Yaskawa INFORM job: A_ROOF_SIDE_0617_2_PAINT_2.JBI

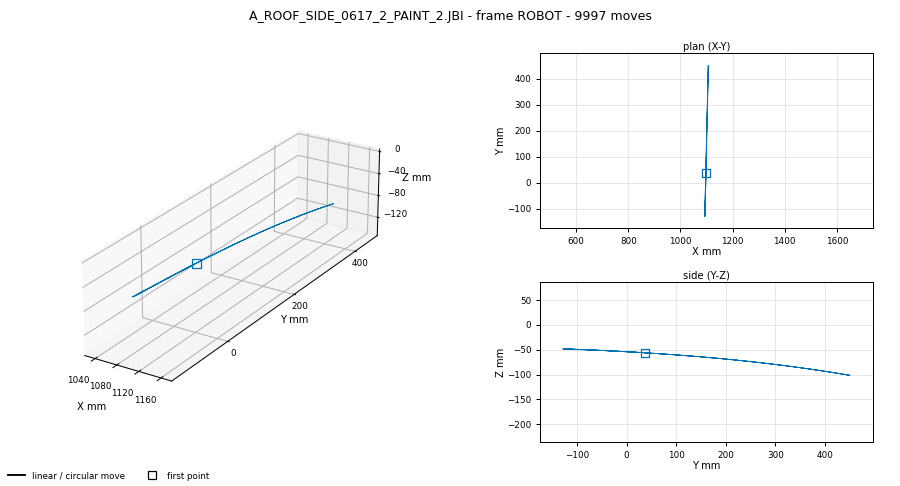
[picture p0: tool path of A_ROOF_SIDE_0617_2_PAINT_2.JBI in frame ROBOT, 9997 of 9997 moves have a stored position in this frame; points joined in program order, loops and branches not executed]
/JOB
//NAME A_ROOF_SIDE_0617_2_PAINT2
//POS
///NPOS 9997,0,0,0,0,0
///TOOL 1
///USER 0
///POSTYPE ROBOT
///RECTAN
///RCONF 1,0,0,0,0,0,0,0,0,0,0,0,0,0,0,0,0,0,0,0,0,0,0,0
C00000=1098.376,37.248,-55.821,176.207,15.311,152.033
C00001=1098.370,36.999,-55.805,176.206,15.311,152.033
C00002=1098.365,36.749,-55.790,176.204,15.310,152.034
C00003=1098.358,36.500,-55.775,176.201,15.310,152.034
C00004=1098.353,36.250,-55.760,176.199,15.308,152.034
C00005=1098.347,36.001,-55.745,176.197,15.308,152.035
C00006=1098.341,35.751,-55.729,176.195,15.307,152.035
C00007=1098.336,35.502,-55.713,176.192,15.306,152.035
C00008=1098.329,35.252,-55.698,176.190,15.306,152.036
C00009=1098.324,35.003,-55.683,176.188,15.305,152.036
C00010=1098.318,34.753,-55.668,176.185,15.304,152.036
C00011=1098.312,34.503,-55.653,176.183,15.303,152.037
C00012=1098.307,34.255,-55.638,176.181,15.303,152.037
C00013=1098.301,34.005,-55.623,176.178,15.302,152.037
C00014=1098.296,33.755,-55.607,176.176,15.301,152.038
C00015=1098.289,33.506,-55.593,176.174,15.301,152.038
C00016=1098.284,33.256,-55.577,176.172,15.300,152.038
C00017=1098.278,33.007,-55.562,176.170,15.299,152.038
C00018=1098.273,32.758,-55.547,176.167,15.298,152.039
C00019=1098.266,32.508,-55.532,176.166,15.298,152.039
C00020=1098.261,32.258,-55.516,176.163,15.296,152.039
C00021=1098.254,31.985,-55.500,176.161,15.296,152.040
C00022=1098.248,31.711,-55.483,176.158,15.295,152.040
C00023=1098.242,31.437,-55.466,176.156,15.294,152.041
C00024=1098.236,31.164,-55.450,176.153,15.293,152.041
C00025=1098.230,30.914,-55.435,176.151,15.292,152.041
C00026=1098.224,30.665,-55.420,176.149,15.292,152.041
C00027=1098.218,30.415,-55.405,176.147,15.291,152.042
C00028=1098.213,30.166,-55.390,176.145,15.290,152.042
C00029=1098.207,29.916,-55.375,176.142,15.290,152.042
C00030=1098.202,29.667,-55.361,176.140,15.288,152.043
C00031=1098.196,29.417,-55.345,176.138,15.288,152.043
C00032=1098.190,29.168,-55.331,176.136,15.287,152.043
C00033=1098.185,28.918,-55.315,176.134,15.287,152.044
C00034=1098.179,28.669,-55.301,176.131,15.285,152.044
C00035=1098.172,28.419,-55.286,176.129,15.285,152.044
C00036=1098.167,28.170,-55.270,176.127,15.284,152.045
C00037=1098.161,27.920,-55.255,176.124,15.283,152.045
C00038=1098.156,27.671,-55.240,176.123,15.282,152.045
C00039=1098.149,27.421,-55.225,176.121,15.281,152.045
C00040=1098.144,27.172,-55.211,176.118,15.281,152.046
C00041=1098.138,26.922,-55.196,176.116,15.280,152.046
C00042=1098.133,26.673,-55.181,176.114,15.279,152.046
C00043=1098.126,26.423,-55.166,176.112,15.278,152.047
C00044=1098.121,26.174,-55.151,176.110,15.278,152.047
C00045=1098.115,25.925,-55.137,176.107,15.277,152.047
C00046=1098.109,25.675,-55.122,176.105,15.276,152.048
C00047=1098.104,25.425,-55.107,176.103,15.275,152.048
C00048=1098.098,25.176,-55.092,176.100,15.274,152.048
C00049=1098.092,24.927,-55.078,176.099,15.274,152.049
C00050=1098.086,24.677,-55.062,176.097,15.273,152.049
C00051=1098.081,24.427,-55.048,176.095,15.272,152.049
C00052=1098.075,24.178,-55.033,176.092,15.271,152.049
C00053=1098.069,23.929,-55.019,176.090,15.271,152.050
C00054=1098.063,23.679,-55.003,176.088,15.270,152.050
C00055=1098.058,23.429,-54.989,176.086,15.269,152.050
C00056=1098.052,23.180,-54.975,176.084,15.268,152.051
C00057=1098.046,22.930,-54.959,176.081,15.268,152.051
C00058=1098.040,22.681,-54.945,176.080,15.267,152.051
C00059=1098.034,22.431,-54.930,176.077,15.265,152.051
C00060=1098.029,22.182,-54.916,176.075,15.265,152.052
C00061=1098.024,21.933,-54.901,176.073,15.264,152.052
C00062=1098.017,21.682,-54.886,176.071,15.264,152.052
C00063=1098.012,21.434,-54.872,176.068,15.262,152.053
C00064=1098.005,21.184,-54.857,176.066,15.262,152.053
C00065=1098.001,20.934,-54.842,176.064,15.261,152.053
C00066=1097.995,20.685,-54.828,176.063,15.260,152.053
C00067=1097.988,20.435,-54.813,176.060,15.259,152.054
C00068=1097.983,20.186,-54.799,176.058,15.258,152.054
C00069=1097.978,19.937,-54.784,176.056,15.258,152.054
C00070=1097.972,19.687,-54.769,176.054,15.257,152.055
C00071=1097.966,19.437,-54.755,176.051,15.256,152.055
C00072=1097.960,19.188,-54.740,176.049,15.255,152.055
C00073=1097.954,18.938,-54.726,176.048,15.254,152.055
C00074=1097.948,18.689,-54.712,176.046,15.254,152.056
C00075=1097.942,18.439,-54.697,176.043,15.253,152.056
C00076=1097.937,18.190,-54.682,176.041,15.252,152.056
C00077=1097.932,17.941,-54.668,176.039,15.251,152.057
C00078=1097.925,17.690,-54.653,176.037,15.251,152.057
C00079=1097.920,17.441,-54.639,176.034,15.249,152.057
C00080=1097.914,17.192,-54.625,176.033,15.248,152.057
C00081=1097.908,16.942,-54.610,176.031,15.248,152.058
C00082=1097.902,16.693,-54.596,176.028,15.247,152.058
C00083=1097.897,16.444,-54.582,176.026,15.246,152.058
C00084=1097.891,16.193,-54.567,176.024,15.245,152.059
C00085=1097.884,15.922,-54.551,176.022,15.245,152.059
C00086=1097.878,15.649,-54.535,176.019,15.243,152.059
C00087=1097.872,15.376,-54.520,176.017,15.243,152.059
C00088=1097.866,15.104,-54.505,176.015,15.241,152.060
C00089=1097.859,14.854,-54.490,176.013,15.241,152.060
C00090=1097.855,14.605,-54.475,176.011,15.240,152.060
C00091=1097.849,14.356,-54.461,176.009,15.240,152.061
C00092=1097.843,14.106,-54.447,176.006,15.238,152.061
C00093=1097.837,13.856,-54.432,176.004,15.237,152.061
C00094=1097.831,13.607,-54.419,176.002,15.237,152.061
C00095=1097.825,13.358,-54.404,176.001,15.236,152.062
C00096=1097.819,13.108,-54.390,175.999,15.235,152.062
C00097=1097.814,12.858,-54.376,175.996,15.234,152.062
C00098=1097.808,12.609,-54.361,175.994,15.234,152.063
C00099=1097.802,12.359,-54.347,175.992,15.233,152.063
C00100=1097.796,12.110,-54.333,175.990,15.232,152.063
C00101=1097.790,11.861,-54.319,175.987,15.231,152.064
C00102=1097.784,11.610,-54.304,175.986,15.230,152.064
C00103=1097.779,11.361,-54.290,175.984,15.229,152.064
C00104=1097.773,11.112,-54.276,175.982,15.229,152.064
C00105=1097.767,10.862,-54.261,175.980,15.228,152.065
C00106=1097.761,10.613,-54.247,175.977,15.227,152.065
C00107=1097.755,10.363,-54.234,175.975,15.226,152.065
C00108=1097.749,10.114,-54.219,175.973,15.225,152.065
C00109=1097.743,9.864,-54.205,175.971,15.225,152.066
C00110=1097.738,9.614,-54.191,175.969,15.224,152.066
C00111=1097.732,9.365,-54.177,175.967,15.223,152.066
C00112=1097.726,9.115,-54.162,175.965,15.222,152.067
C00113=1097.720,8.866,-54.149,175.963,15.221,152.067
C00114=1097.715,8.616,-54.135,175.961,15.221,152.067
C00115=1097.708,8.367,-54.121,175.958,15.219,152.067
C00116=1097.702,8.117,-54.107,175.957,15.219,152.068
C00117=1097.697,7.868,-54.093,175.955,15.218,152.068
C00118=1097.691,7.618,-54.079,175.953,15.217,152.068
C00119=1097.685,7.369,-54.064,175.951,15.216,152.068
C00120=1097.679,7.119,-54.050,175.948,15.215,152.069
C00121=1097.674,6.869,-54.036,175.946,15.214,152.069
C00122=1097.668,6.620,-54.023,175.944,15.214,152.069
C00123=1097.662,6.370,-54.009,175.943,15.213,152.069
C00124=1097.656,6.121,-53.994,175.941,15.212,152.070
C00125=1097.650,5.871,-53.980,175.938,15.211,152.070
C00126=1097.645,5.622,-53.966,175.936,15.210,152.070
C00127=1097.639,5.372,-53.952,175.934,15.209,152.070
C00128=1097.633,5.123,-53.939,175.932,15.209,152.071
C00129=1097.627,4.874,-53.925,175.931,15.208,152.071
C00130=1097.621,4.623,-53.910,175.928,15.207,152.071
C00131=1097.616,4.374,-53.896,175.926,15.206,152.072
C00132=1097.610,4.124,-53.883,175.924,15.205,152.072
C00133=1097.604,3.875,-53.869,175.922,15.204,152.072
C00134=1097.599,3.625,-53.855,175.920,15.204,152.072
C00135=1097.593,3.376,-53.842,175.918,15.202,152.073
C00136=1097.588,3.126,-53.828,175.916,15.202,152.073
C00137=1097.581,2.877,-53.813,175.914,15.201,152.073
C00138=1097.575,2.627,-53.800,175.912,15.200,152.073
C00139=1097.570,2.378,-53.786,175.910,15.199,152.073
C00140=1097.564,2.128,-53.772,175.908,15.198,152.074
C00141=1097.559,1.879,-53.758,175.906,15.197,152.074
C00142=1097.553,1.629,-53.745,175.904,15.196,152.074
C00143=1097.547,1.380,-53.731,175.902,15.195,152.075
C00144=1097.541,1.130,-53.717,175.900,15.195,152.075
C00145=1097.536,0.880,-53.703,175.898,15.194,152.075
C00146=1097.529,0.631,-53.689,175.896,15.193,152.075
C00147=1097.524,0.381,-53.676,175.894,15.192,152.076
C00148=1097.518,0.132,-53.662,175.892,15.191,152.076
C00149=1097.512,-0.139,-53.646,175.890,15.190,152.076
C00150=1097.506,-0.409,-53.632,175.887,15.189,152.076
C00151=1097.500,-0.679,-53.617,175.886,15.188,152.077
C00152=1097.493,-0.949,-53.602,175.884,15.188,152.077
C00153=1097.488,-1.199,-53.589,175.881,15.186,152.077
C00154=1097.482,-1.448,-53.575,175.879,15.185,152.077
C00155=1097.476,-1.699,-53.560,175.878,15.184,152.078
C00156=1097.470,-1.948,-53.547,175.876,15.184,152.078
C00157=1097.465,-2.198,-53.534,175.874,15.183,152.078
C00158=1097.459,-2.448,-53.520,175.871,15.182,152.078
C00159=1097.454,-2.697,-53.506,175.869,15.181,152.079
C00160=1097.448,-2.946,-53.493,175.867,15.180,152.079
C00161=1097.442,-3.196,-53.479,175.866,15.179,152.079
C00162=1097.437,-3.446,-53.465,175.864,15.178,152.079
C00163=1097.431,-3.695,-53.452,175.862,15.177,152.079
C00164=1097.425,-3.944,-53.438,175.859,15.176,152.080
C00165=1097.419,-4.194,-53.425,175.858,15.175,152.080
C00166=1097.413,-4.443,-53.411,175.856,15.175,152.080
C00167=1097.407,-4.693,-53.398,175.854,15.174,152.081
C00168=1097.401,-4.943,-53.384,175.852,15.173,152.081
C00169=1097.395,-5.193,-53.371,175.850,15.172,152.081
C00170=1097.390,-5.442,-53.357,175.847,15.171,152.081
C00171=1097.383,-5.692,-53.344,175.845,15.170,152.082
C00172=1097.378,-5.941,-53.330,175.844,15.170,152.082
C00173=1097.372,-6.190,-53.317,175.842,15.169,152.082
C00174=1097.367,-6.441,-53.304,175.840,15.168,152.082
C00175=1097.360,-6.690,-53.290,175.838,15.167,152.082
C00176=1097.355,-6.939,-53.276,175.836,15.166,152.083
C00177=1097.349,-7.189,-53.263,175.834,15.165,152.083
C00178=1097.343,-7.438,-53.249,175.832,15.164,152.083
C00179=1097.337,-7.688,-53.237,175.830,15.163,152.084
C00180=1097.331,-7.937,-53.223,175.828,15.163,152.084
C00181=1097.326,-8.187,-53.210,175.826,15.162,152.084
C00182=1097.319,-8.436,-53.196,175.824,15.161,152.084
C00183=1097.314,-8.686,-53.183,175.822,15.161,152.085
C00184=1097.308,-8.936,-53.170,175.820,15.159,152.085
C00185=1097.303,-9.185,-53.156,175.818,15.158,152.085
C00186=1097.296,-9.435,-53.143,175.816,15.157,152.085
C00187=1097.291,-9.685,-53.130,175.814,15.157,152.085
C00188=1097.284,-9.935,-53.116,175.813,15.156,152.086
C00189=1097.278,-10.184,-53.103,175.811,15.155,152.086
C00190=1097.273,-10.434,-53.089,175.809,15.154,152.086
C00191=1097.267,-10.683,-53.077,175.806,15.153,152.087
C00192=1097.262,-10.932,-53.063,175.805,15.152,152.087
C00193=1097.256,-11.182,-53.050,175.803,15.151,152.087
C00194=1097.251,-11.432,-53.036,175.801,15.150,152.087
C00195=1097.244,-11.681,-53.023,175.799,15.150,152.087
C00196=1097.238,-11.930,-53.010,175.797,15.149,152.088
C00197=1097.233,-12.180,-52.997,175.795,15.148,152.088
C00198=1097.227,-12.430,-52.983,175.794,15.147,152.088
C00199=1097.222,-12.680,-52.970,175.791,15.146,152.088
C00200=1097.215,-12.929,-52.957,175.789,15.145,152.089
C00201=1097.209,-13.178,-52.944,175.787,15.144,152.089
C00202=1097.204,-13.429,-52.931,175.785,15.143,152.089
C00203=1097.198,-13.678,-52.917,175.783,15.143,152.089
C00204=1097.193,-13.928,-52.904,175.782,15.142,152.089
C00205=1097.186,-14.177,-52.891,175.780,15.141,152.090
C00206=1097.180,-14.427,-52.878,175.778,15.140,152.090
C00207=1097.175,-14.677,-52.865,175.775,15.139,152.090
C00208=1097.169,-14.926,-52.851,175.773,15.138,152.091
C00209=1097.163,-15.176,-52.839,175.772,15.137,152.091
C00210=1097.157,-15.426,-52.825,175.770,15.136,152.091
C00211=1097.151,-15.675,-52.812,175.768,15.135,152.091
C00212=1097.145,-15.925,-52.799,175.766,15.135,152.091
C00213=1097.139,-16.194,-52.785,175.764,15.134,152.092
C00214=1097.133,-16.462,-52.771,175.762,15.133,152.092
C00215=1097.127,-16.731,-52.757,175.760,15.132,152.092
C00216=1097.120,-16.999,-52.743,175.758,15.131,152.092
C00217=1097.114,-17.249,-52.730,175.756,15.130,152.093
C00218=1097.109,-17.498,-52.716,175.754,15.129,152.093
C00219=1097.103,-17.748,-52.704,175.752,15.128,152.093
C00220=1097.097,-17.997,-52.691,175.750,15.127,152.093
C00221=1097.091,-18.247,-52.678,175.748,15.126,152.094
C00222=1097.085,-18.497,-52.665,175.746,15.126,152.094
C00223=1097.079,-18.747,-52.652,175.744,15.125,152.094
C00224=1097.073,-18.997,-52.639,175.743,15.124,152.094
C00225=1097.067,-19.246,-52.626,175.741,15.123,152.094
C00226=1097.061,-19.496,-52.613,175.739,15.122,152.095
C00227=1097.056,-19.744,-52.600,175.737,15.122,152.095
C00228=1097.050,-19.994,-52.588,175.735,15.121,152.095
C00229=1097.044,-20.244,-52.574,175.733,15.120,152.096
C00230=1097.038,-20.494,-52.561,175.731,15.118,152.096
C00231=1097.033,-20.743,-52.549,175.729,15.118,152.096
C00232=1097.026,-20.993,-52.536,175.727,15.117,152.096
C00233=1097.020,-21.243,-52.523,175.725,15.116,152.096
C00234=1097.014,-21.492,-52.510,175.723,15.115,152.097
C00235=1097.010,-21.741,-52.497,175.722,15.114,152.097
C00236=1097.004,-21.991,-52.484,175.720,15.114,152.097
C00237=1096.998,-22.241,-52.471,175.718,15.113,152.097
C00238=1096.992,-22.490,-52.459,175.716,15.112,152.098
C00239=1096.986,-22.740,-52.446,175.714,15.111,152.098
C00240=1096.979,-22.990,-52.433,175.713,15.110,152.098
C00241=1096.974,-23.239,-52.420,175.710,15.109,152.098
C00242=1096.969,-23.489,-52.407,175.708,15.108,152.098
C00243=1096.963,-23.738,-52.394,175.706,15.107,152.099
C00244=1096.957,-23.988,-52.382,175.704,15.107,152.099
C00245=1096.951,-24.238,-52.369,175.703,15.105,152.099
C00246=1096.945,-24.488,-52.356,175.701,15.105,152.099
C00247=1096.939,-24.736,-52.344,175.699,15.104,152.100
C00248=1096.934,-24.986,-52.331,175.697,15.103,152.100
C00249=1096.928,-25.236,-52.318,175.696,15.102,152.100
C00250=1096.921,-25.485,-52.305,175.694,15.101,152.100
C00251=1096.916,-25.735,-52.293,175.692,15.101,152.100
C00252=1096.911,-25.985,-52.280,175.690,15.100,152.101
C00253=1096.905,-26.235,-52.267,175.688,15.099,152.101
C00254=1096.899,-26.484,-52.254,175.686,15.097,152.101
C00255=1096.893,-26.734,-52.241,175.684,15.097,152.101
C00256=1096.887,-26.984,-52.229,175.682,15.096,152.102
C00257=1096.882,-27.233,-52.217,175.680,15.095,152.102
C00258=1096.876,-27.483,-52.204,175.679,15.094,152.102
C00259=1096.870,-27.732,-52.191,175.677,15.093,152.102
C00260=1096.864,-27.982,-52.178,175.675,15.093,152.103
C00261=1096.858,-28.232,-52.166,175.673,15.092,152.103
C00262=1096.851,-28.481,-52.154,175.671,15.091,152.103
C00263=1096.846,-28.731,-52.142,175.669,15.090,152.103
C00264=1096.840,-28.980,-52.128,175.668,15.089,152.103
C00265=1096.834,-29.230,-52.116,175.666,15.088,152.104
C00266=1096.828,-29.480,-52.103,175.664,15.088,152.104
C00267=1096.822,-29.729,-52.091,175.662,15.087,152.104
C00268=1096.817,-29.979,-52.079,175.660,15.086,152.104
C00269=1096.811,-30.229,-52.066,175.658,15.085,152.105
C00270=1096.805,-30.478,-52.053,175.657,15.084,152.105
C00271=1096.799,-30.728,-52.040,175.655,15.084,152.105
C00272=1096.793,-30.977,-52.028,175.653,15.083,152.105
C00273=1096.787,-31.226,-52.016,175.650,15.082,152.106
C00274=1096.781,-31.476,-52.003,175.649,15.080,152.106
C00275=1096.775,-31.726,-51.991,175.647,15.080,152.106
C00276=1096.769,-31.976,-51.978,175.645,15.079,152.106
C00277=1096.763,-32.244,-51.965,175.643,15.078,152.106
C00278=1096.757,-32.511,-51.952,175.641,15.078,152.107
C00279=1096.750,-32.780,-51.938,175.639,15.077,152.107
C00280=1096.744,-33.047,-51.924,175.638,15.076,152.107
C00281=1096.737,-33.297,-51.912,175.636,15.075,152.107
C00282=1096.732,-33.546,-51.900,175.634,15.074,152.108
C00283=1096.726,-33.796,-51.888,175.632,15.073,152.108
C00284=1096.720,-34.046,-51.875,175.629,15.072,152.108
C00285=1096.714,-34.296,-51.863,175.628,15.071,152.108
C00286=1096.709,-34.545,-51.850,175.626,15.070,152.109
C00287=1096.702,-34.794,-51.838,175.624,15.069,152.109
C00288=1096.697,-35.044,-51.826,175.622,15.069,152.109
C00289=1096.691,-35.294,-51.814,175.620,15.068,152.109
C00290=1096.685,-35.543,-51.801,175.619,15.067,152.109
C00291=1096.679,-35.793,-51.789,175.617,15.066,152.110
C00292=1096.674,-36.042,-51.776,175.615,15.065,152.110
C00293=1096.668,-36.292,-51.764,175.613,15.064,152.110
C00294=1096.662,-36.542,-51.752,175.611,15.063,152.110
C00295=1096.657,-36.792,-51.740,175.609,15.063,152.111
C00296=1096.651,-37.042,-51.728,175.608,15.062,152.111
C00297=1096.645,-37.292,-51.715,175.606,15.061,152.111
C00298=1096.639,-37.541,-51.703,175.604,15.060,152.111
C00299=1096.633,-37.790,-51.691,175.602,15.059,152.111
C00300=1096.627,-38.040,-51.679,175.600,15.059,152.112
C00301=1096.622,-38.289,-51.666,175.599,15.058,152.112
C00302=1096.616,-38.539,-51.654,175.597,15.057,152.112
C00303=1096.609,-38.789,-51.642,175.595,15.056,152.112
C00304=1096.604,-39.038,-51.630,175.593,15.055,152.113
C00305=1096.598,-39.288,-51.617,175.591,15.055,152.113
C00306=1096.592,-39.538,-51.606,175.590,15.053,152.113
C00307=1096.586,-39.787,-51.594,175.588,15.053,152.113
C00308=1096.580,-40.037,-51.581,175.586,15.052,152.113
C00309=1096.574,-40.287,-51.569,175.584,15.051,152.114
C00310=1096.568,-40.537,-51.557,175.582,15.050,152.114
C00311=1096.562,-40.786,-51.545,175.580,15.050,152.114
C00312=1096.556,-41.035,-51.533,175.579,15.049,152.114
C00313=1096.550,-41.286,-51.521,175.577,15.048,152.115
C00314=1096.545,-41.535,-51.509,175.575,15.047,152.115
C00315=1096.538,-41.785,-51.497,175.573,15.046,152.115
C00316=1096.533,-42.034,-51.484,175.571,15.046,152.115
C00317=1096.526,-42.283,-51.472,175.570,15.044,152.116
C00318=1096.521,-42.534,-51.461,175.568,15.044,152.116
C00319=1096.515,-42.783,-51.448,175.566,15.043,152.116
C00320=1096.509,-43.033,-51.436,175.564,15.042,152.116
C00321=1096.503,-43.282,-51.424,175.562,15.042,152.117
C00322=1096.497,-43.531,-51.412,175.561,15.040,152.117
C00323=1096.491,-43.782,-51.400,175.559,15.040,152.117
C00324=1096.485,-44.032,-51.388,175.557,15.039,152.117
C00325=1096.479,-44.281,-51.376,175.555,15.038,152.117
C00326=1096.473,-44.530,-51.364,175.553,15.037,152.118
C00327=1096.468,-44.780,-51.353,175.551,15.036,152.118
C00328=1096.462,-45.030,-51.340,175.550,15.036,152.118
C00329=1096.456,-45.280,-51.328,175.548,15.035,152.118
C00330=1096.450,-45.529,-51.317,175.546,15.034,152.119
C00331=1096.444,-45.779,-51.304,175.545,15.034,152.119
C00332=1096.438,-46.028,-51.293,175.543,15.033,152.119
C00333=1096.432,-46.278,-51.280,175.541,15.032,152.119
C00334=1096.426,-46.528,-51.269,175.539,15.031,152.119
C00335=1096.420,-46.777,-51.257,175.537,15.031,152.120
C00336=1096.414,-47.027,-51.245,175.536,15.029,152.120
C00337=1096.409,-47.277,-51.233,175.534,15.029,152.120
C00338=1096.403,-47.526,-51.221,175.532,15.028,152.120
C00339=1096.397,-47.775,-51.209,175.530,15.027,152.121
C00340=1096.391,-48.026,-51.197,175.529,15.026,152.121
C00341=1096.385,-48.293,-51.185,175.527,15.025,152.121
C00342=1096.378,-48.562,-51.172,175.525,15.025,152.121
C00343=1096.372,-48.830,-51.160,175.523,15.024,152.121
C00344=1096.366,-49.098,-51.147,175.520,15.023,152.122
C00345=1096.360,-49.348,-51.134,175.518,15.022,152.122
C00346=1096.354,-49.598,-51.123,175.518,15.021,152.122
C00347=1096.348,-49.848,-51.111,175.516,15.021,152.122
C00348=1096.343,-50.097,-51.100,175.514,15.020,152.123
C00349=1096.337,-50.347,-51.087,175.512,15.019,152.123
C00350=1096.331,-50.596,-51.076,175.510,15.018,152.123
C00351=1096.324,-50.846,-51.065,175.509,15.017,152.123
C00352=1096.319,-51.096,-51.052,175.507,15.017,152.123
C00353=1096.313,-51.345,-51.041,175.505,15.016,152.124
C00354=1096.306,-51.595,-51.029,175.503,15.015,152.124
C00355=1096.301,-51.845,-51.018,175.501,15.014,152.124
C00356=1096.294,-52.094,-51.006,175.499,15.014,152.125
C00357=1096.288,-52.344,-50.994,175.498,15.012,152.125
C00358=1096.283,-52.594,-50.982,175.496,15.012,152.125
C00359=1096.276,-52.843,-50.970,175.494,15.011,152.125
C00360=1096.270,-53.093,-50.959,175.492,15.010,152.125
C00361=1096.264,-53.342,-50.948,175.490,15.010,152.126
C00362=1096.259,-53.592,-50.936,175.489,15.009,152.126
C00363=1096.252,-53.842,-50.924,175.487,15.009,152.126
C00364=1096.246,-54.092,-50.913,175.485,15.008,152.126
C00365=1096.240,-54.341,-50.901,175.484,15.007,152.127
C00366=1096.234,-54.591,-50.889,175.482,15.006,152.127
C00367=1096.228,-54.840,-50.878,175.480,15.005,152.127
C00368=1096.222,-55.090,-50.867,175.478,15.005,152.127
C00369=1096.216,-55.340,-50.854,175.476,15.004,152.128
C00370=1096.210,-55.590,-50.843,175.474,15.003,152.128
C00371=1096.204,-55.839,-50.832,175.472,15.003,152.128
C00372=1096.198,-56.089,-50.820,175.471,15.001,152.128
C00373=1096.193,-56.339,-50.809,175.469,15.001,152.128
C00374=1096.186,-56.588,-50.797,175.468,15.001,152.129
C00375=1096.180,-56.838,-50.786,175.466,15.000,152.129
C00376=1096.174,-57.087,-50.774,175.464,14.999,152.129
C00377=1096.168,-57.337,-50.763,175.462,14.998,152.129
C00378=1096.162,-57.587,-50.751,175.460,14.998,152.130
C00379=1096.156,-57.836,-50.740,175.459,14.996,152.130
C00380=1096.150,-58.086,-50.728,175.457,14.996,152.130
C00381=1096.144,-58.336,-50.718,175.455,14.995,152.130
C00382=1096.138,-58.586,-50.705,175.453,14.994,152.131
C00383=1096.133,-58.835,-50.694,175.451,14.994,152.131
C00384=1096.126,-59.085,-50.682,175.450,14.993,152.131
C00385=1096.120,-59.334,-50.671,175.448,14.993,152.131
C00386=1096.114,-59.584,-50.660,175.446,14.992,152.131
C00387=1096.109,-59.834,-50.648,175.445,14.991,152.132
C00388=1096.102,-60.084,-50.637,175.443,14.990,152.132
C00389=1096.096,-60.333,-50.626,175.441,14.989,152.132
C00390=1096.090,-60.583,-50.614,175.439,14.989,152.133
C00391=1096.084,-60.832,-50.603,175.437,14.988,152.133
C00392=1096.079,-61.082,-50.591,175.435,14.987,152.133
C00393=1096.072,-61.332,-50.580,175.434,14.987,152.133
C00394=1096.067,-61.581,-50.569,175.432,14.986,152.133
C00395=1096.060,-61.831,-50.557,175.431,14.985,152.134
C00396=1096.055,-62.081,-50.547,175.429,14.985,152.134
C00397=1096.048,-62.330,-50.535,175.427,14.984,152.134
C00398=1096.043,-62.580,-50.523,175.425,14.983,152.134
C00399=1096.037,-62.830,-50.512,175.423,14.982,152.135
C00400=1096.031,-63.080,-50.501,175.421,14.981,152.135
C00401=1096.025,-63.329,-50.489,175.420,14.981,152.135
C00402=1096.019,-63.579,-50.478,175.418,14.980,152.135
C00403=1096.013,-63.828,-50.467,175.417,14.980,152.136
C00404=1096.007,-64.078,-50.456,175.415,14.979,152.136
C00405=1096.000,-64.348,-50.443,175.413,14.978,152.136
C00406=1095.994,-64.618,-50.431,175.411,14.977,152.136
C00407=1095.988,-64.887,-50.419,175.409,14.976,152.136
C00408=1095.982,-65.157,-50.407,175.407,14.976,152.137
C00409=1095.976,-65.406,-50.396,175.406,14.975,152.137
C00410=1095.969,-65.656,-50.384,175.404,14.974,152.137
C00411=1095.964,-65.905,-50.374,175.402,14.973,152.138
C00412=1095.957,-66.155,-50.362,175.400,14.973,152.138
C00413=1095.951,-66.405,-50.351,175.399,14.973,152.138
C00414=1095.946,-66.655,-50.340,175.397,14.971,152.138
C00415=1095.940,-66.904,-50.328,175.395,14.971,152.138
C00416=1095.934,-67.154,-50.317,175.394,14.970,152.139
C00417=1095.928,-67.403,-50.306,175.392,14.969,152.139
C00418=1095.922,-67.653,-50.295,175.390,14.969,152.139
C00419=1095.916,-67.903,-50.284,175.388,14.968,152.139
C00420=1095.910,-68.152,-50.273,175.387,14.967,152.139
C00421=1095.904,-68.403,-50.262,175.385,14.967,152.140
C00422=1095.898,-68.652,-50.251,175.383,14.966,152.140
C00423=1095.893,-68.902,-50.240,175.381,14.965,152.140
C00424=1095.886,-69.151,-50.228,175.380,14.964,152.141
C00425=1095.881,-69.401,-50.217,175.378,14.964,152.141
C00426=1095.875,-69.650,-50.206,175.377,14.964,152.141
C00427=1095.870,-69.900,-50.195,175.375,14.962,152.141
C00428=1095.863,-70.150,-50.184,175.373,14.962,152.141
C00429=1095.857,-70.400,-50.173,175.371,14.961,152.142
C00430=1095.852,-70.649,-50.162,175.369,14.960,152.142
C00431=1095.845,-70.899,-50.151,175.367,14.960,152.142
C00432=1095.840,-71.149,-50.140,175.366,14.959,152.142
C00433=1095.834,-71.398,-50.129,175.364,14.959,152.143
C00434=1095.828,-71.648,-50.118,175.363,14.958,152.143
C00435=1095.822,-71.898,-50.107,175.361,14.957,152.143
C00436=1095.816,-72.147,-50.096,175.359,14.956,152.143
C00437=1095.810,-72.397,-50.085,175.357,14.955,152.144
C00438=1095.805,-72.646,-50.074,175.355,14.955,152.144
C00439=1095.798,-72.897,-50.063,175.354,14.955,152.144
C00440=1095.793,-73.146,-50.052,175.353,14.953,152.144
C00441=1095.787,-73.396,-50.041,175.351,14.953,152.144
C00442=1095.781,-73.645,-50.031,175.349,14.952,152.145
C00443=1095.775,-73.895,-50.019,175.347,14.951,152.145
C00444=1095.769,-74.145,-50.008,175.346,14.951,152.145
C00445=1095.763,-74.394,-49.998,175.344,14.950,152.145
C00446=1095.757,-74.644,-49.986,175.342,14.950,152.146
C00447=1095.751,-74.894,-49.975,175.340,14.949,152.146
C00448=1095.745,-75.143,-49.965,175.338,14.948,152.146
C00449=1095.740,-75.393,-49.954,175.337,14.948,152.146
C00450=1095.733,-75.643,-49.942,175.336,14.947,152.147
C00451=1095.728,-75.893,-49.932,175.334,14.946,152.147
C00452=1095.721,-76.142,-49.922,175.332,14.946,152.147
C00453=1095.715,-76.393,-49.911,175.330,14.945,152.147
C00454=1095.709,-76.642,-49.900,175.329,14.945,152.148
C00455=1095.704,-76.892,-49.889,175.327,14.944,152.148
C00456=1095.698,-77.141,-49.878,175.325,14.943,152.148
C00457=1095.692,-77.391,-49.867,175.323,14.943,152.148
C00458=1095.685,-77.640,-49.857,175.321,14.942,152.149
C00459=1095.679,-77.890,-49.846,175.320,14.942,152.149
C00460=1095.674,-78.139,-49.835,175.318,14.941,152.149
C00461=1095.668,-78.390,-49.824,175.316,14.940,152.149
C00462=1095.662,-78.640,-49.813,175.315,14.940,152.150
C00463=1095.656,-78.889,-49.803,175.313,14.939,152.150
C00464=1095.650,-79.138,-49.792,175.312,14.939,152.150
C00465=1095.643,-79.389,-49.781,175.310,14.938,152.150
C00466=1095.637,-79.638,-49.770,175.308,14.937,152.151
C00467=1095.632,-79.888,-49.759,175.306,14.936,152.151
C00468=1095.626,-80.138,-49.749,175.305,14.936,152.151
C00469=1095.619,-80.409,-49.738,175.303,14.936,152.151
C00470=1095.612,-80.681,-49.726,175.301,14.935,152.152
C00471=1095.606,-80.953,-49.714,175.299,14.934,152.152
C00472=1095.599,-81.224,-49.702,175.297,14.934,152.152
C00473=1095.593,-81.474,-49.693,175.295,14.933,152.153
C00474=1095.587,-81.724,-49.682,175.293,14.932,152.153
C00475=1095.581,-81.974,-49.670,175.292,14.932,152.153
C00476=1095.574,-82.223,-49.660,175.290,14.932,152.153
C00477=1095.569,-82.473,-49.649,175.289,14.931,152.154
C00478=1095.563,-82.723,-49.639,175.287,14.930,152.154
C00479=1095.556,-82.973,-49.628,175.286,14.930,152.154
C00480=1095.550,-83.222,-49.618,175.284,14.929,152.154
C00481=1095.544,-83.471,-49.607,175.282,14.929,152.155
C00482=1095.539,-83.721,-49.597,175.280,14.928,152.155
C00483=1095.532,-83.972,-49.586,175.279,14.928,152.155
C00484=1095.526,-84.221,-49.576,175.277,14.927,152.155
C00485=1095.520,-84.470,-49.565,175.275,14.926,152.156
C00486=1095.515,-84.720,-49.555,175.273,14.926,152.156
C00487=1095.508,-84.970,-49.544,175.272,14.926,152.156
C00488=1095.502,-85.220,-49.533,175.270,14.925,152.156
C00489=1095.496,-85.470,-49.523,175.268,14.924,152.157
C00490=1095.490,-85.719,-49.513,175.266,14.923,152.157
C00491=1095.484,-85.968,-49.502,175.265,14.923,152.157
C00492=1095.477,-86.219,-49.492,175.263,14.923,152.157
C00493=1095.472,-86.468,-49.481,175.262,14.922,152.158
C00494=1095.465,-86.718,-49.471,175.260,14.921,152.158
C00495=1095.460,-86.968,-49.460,175.259,14.921,152.158
C00496=1095.454,-87.217,-49.450,175.256,14.921,152.159
C00497=1095.447,-87.466,-49.439,175.254,14.920,152.159
C00498=1095.441,-87.717,-49.429,175.253,14.919,152.159
C00499=1095.435,-87.966,-49.418,175.251,14.919,152.159
C00500=1095.429,-88.216,-49.408,175.250,14.919,152.160
C00501=1095.423,-88.466,-49.398,175.248,14.918,152.160
C00502=1095.417,-88.715,-49.387,175.247,14.918,152.160
C00503=1095.412,-88.965,-49.377,175.245,14.917,152.160
C00504=1095.405,-89.215,-49.366,175.243,14.916,152.161
C00505=1095.399,-89.465,-49.355,175.241,14.916,152.161
C00506=1095.393,-89.714,-49.346,175.240,14.916,152.161
C00507=1095.387,-89.964,-49.335,175.238,14.915,152.161
C00508=1095.381,-90.214,-49.325,175.236,14.914,152.162
C00509=1095.375,-90.463,-49.315,175.235,14.914,152.162
C00510=1095.369,-90.712,-49.304,175.233,14.913,152.162
C00511=1095.363,-90.963,-49.294,175.231,14.913,152.162
C00512=1095.356,-91.212,-49.284,175.229,14.912,152.163
C00513=1095.351,-91.463,-49.273,175.228,14.912,152.163
C00514=1095.345,-91.712,-49.262,175.226,14.911,152.163
C00515=1095.339,-91.962,-49.253,175.224,14.910,152.163
C00516=1095.333,-92.211,-49.242,175.223,14.910,152.164
C00517=1095.327,-92.461,-49.232,175.221,14.910,152.164
C00518=1095.321,-92.711,-49.222,175.219,14.909,152.164
C00519=1095.315,-92.960,-49.212,175.217,14.909,152.165
C00520=1095.309,-93.211,-49.201,175.216,14.909,152.165
C00521=1095.303,-93.460,-49.191,175.214,14.908,152.165
C00522=1095.297,-93.710,-49.180,175.212,14.907,152.165
C00523=1095.291,-93.960,-49.171,175.211,14.907,152.166
C00524=1095.285,-94.209,-49.160,175.209,14.906,152.166
C00525=1095.279,-94.459,-49.150,175.208,14.906,152.166
C00526=1095.273,-94.708,-49.139,175.206,14.906,152.166
C00527=1095.267,-94.958,-49.130,175.205,14.905,152.167
C00528=1095.261,-95.208,-49.119,175.203,14.904,152.167
C00529=1095.255,-95.458,-49.109,175.202,14.904,152.167
C00530=1095.249,-95.708,-49.099,175.200,14.903,152.167
C00531=1095.243,-95.957,-49.089,175.198,14.903,152.168
C00532=1095.238,-96.207,-49.079,175.196,14.902,152.168
C00533=1095.231,-96.481,-49.068,175.194,14.902,152.168
C00534=1095.224,-96.755,-49.057,175.193,14.902,152.169
C00535=1095.218,-97.028,-49.045,175.191,14.901,152.169
C00536=1095.211,-97.302,-49.034,175.189,14.900,152.169
C00537=1095.204,-97.553,-49.024,175.187,14.899,152.169
C00538=1095.199,-97.803,-49.014,175.186,14.899,152.170
C00539=1095.192,-98.052,-49.003,175.184,14.899,152.170
C00540=1095.186,-98.302,-48.994,175.182,14.898,152.170
C00541=1095.180,-98.551,-48.983,175.181,14.898,152.170
C00542=1095.174,-98.801,-48.973,175.179,14.898,152.171
C00543=1095.168,-99.051,-48.964,175.177,14.897,152.171
C00544=1095.162,-99.300,-48.953,175.176,14.897,152.171
C00545=1095.156,-99.550,-48.943,175.173,14.897,152.172
C00546=1095.150,-99.800,-48.934,175.172,14.896,152.172
C00547=1095.144,-100.050,-48.923,175.170,14.896,152.172
C00548=1095.138,-100.299,-48.913,175.169,14.895,152.172
C00549=1095.132,-100.549,-48.904,175.167,14.894,152.173
C00550=1095.125,-100.798,-48.894,175.166,14.894,152.173
C00551=1095.119,-101.049,-48.883,175.163,14.894,152.173
C00552=1095.113,-101.299,-48.874,175.162,14.894,152.174
C00553=1095.107,-101.548,-48.863,175.160,14.893,152.174
C00554=1095.101,-101.798,-48.853,175.159,14.893,152.174
C00555=1095.095,-102.048,-48.843,175.157,14.892,152.174
C00556=1095.089,-102.297,-48.833,175.156,14.892,152.175
C00557=1095.083,-102.547,-48.824,175.153,14.892,152.175
C00558=1095.077,-102.797,-48.813,175.152,14.891,152.175
C00559=1095.071,-103.047,-48.804,175.150,14.891,152.176
C00560=1095.064,-103.296,-48.794,175.148,14.890,152.176
C00561=1095.058,-103.546,-48.784,175.147,14.890,152.176
C00562=1095.053,-103.796,-48.774,175.145,14.890,152.176
C00563=1095.046,-104.045,-48.764,175.144,14.890,152.177
C00564=1095.040,-104.295,-48.754,175.142,14.889,152.177
C00565=1095.034,-104.545,-48.744,175.140,14.888,152.177
C00566=1095.029,-104.795,-48.734,175.139,14.888,152.177
C00567=1095.022,-105.045,-48.725,175.137,14.888,152.178
C00568=1095.016,-105.294,-48.714,175.135,14.887,152.178
C00569=1095.010,-105.544,-48.705,175.134,14.887,152.178
C00570=1095.004,-105.794,-48.695,175.132,14.886,152.179
C00571=1094.998,-106.044,-48.685,175.131,14.886,152.179
C00572=1094.992,-106.293,-48.675,175.129,14.886,152.179
C00573=1094.986,-106.543,-48.665,175.127,14.885,152.180
C00574=1094.979,-106.792,-48.656,175.126,14.885,152.180
C00575=1094.974,-107.042,-48.646,175.124,14.885,152.180
C00576=1094.968,-107.292,-48.636,175.122,14.884,152.180
C00577=1094.962,-107.542,-48.626,175.121,14.884,152.181
C00578=1094.955,-107.791,-48.616,175.119,14.884,152.181
C00579=1094.949,-108.041,-48.607,175.118,14.884,152.181
C00580=1094.943,-108.291,-48.597,175.116,14.883,152.181
C00581=1094.937,-108.541,-48.587,175.113,14.883,152.182
C00582=1094.931,-108.791,-48.577,175.112,14.882,152.182
C00583=1094.925,-109.041,-48.568,175.110,14.882,152.182
C00584=1094.918,-109.290,-48.557,175.109,14.882,152.183
C00585=1094.912,-109.540,-48.548,175.107,14.881,152.183
C00586=1094.906,-109.789,-48.538,175.105,14.881,152.183
C00587=1094.900,-110.039,-48.529,175.104,14.881,152.184
C00588=1094.894,-110.289,-48.519,175.102,14.880,152.184
C00589=1094.888,-110.539,-48.510,175.101,14.880,152.184
C00590=1094.881,-110.788,-48.500,175.099,14.880,152.184
C00591=1094.876,-111.038,-48.491,175.097,14.879,152.185
C00592=1094.870,-111.287,-48.481,175.096,14.879,152.185
C00593=1094.864,-111.537,-48.470,175.094,14.879,152.185
C00594=1094.858,-111.787,-48.461,175.093,14.879,152.186
C00595=1094.852,-112.036,-48.451,175.090,14.878,152.186
C00596=1094.845,-112.286,-48.442,175.089,14.878,152.186
C00597=1094.839,-112.551,-48.432,175.087,14.878,152.187
C00598=1094.833,-112.816,-48.421,175.085,14.877,152.187
C00599=1094.826,-113.081,-48.412,175.084,14.877,152.187
C00600=1094.820,-113.345,-48.402,175.082,14.877,152.187
C00601=1094.813,-113.595,-48.392,175.080,14.876,152.188
C00602=1094.807,-113.844,-48.382,175.079,14.876,152.188
C00603=1094.801,-114.094,-48.372,175.077,14.876,152.188
C00604=1094.795,-114.344,-48.363,175.076,14.876,152.189
C00605=1094.788,-114.594,-48.353,175.074,14.875,152.189
C00606=1094.782,-114.844,-48.344,175.072,14.875,152.189
C00607=1094.776,-115.093,-48.334,175.070,14.875,152.190
C00608=1094.770,-115.343,-48.325,175.068,14.874,152.190
C00609=1094.764,-115.593,-48.315,175.067,14.874,152.190
C00610=1094.758,-115.843,-48.305,175.065,14.874,152.191
C00611=1094.751,-116.093,-48.296,175.064,14.874,152.191
C00612=1094.746,-116.342,-48.287,175.062,14.873,152.191
C00613=1094.740,-116.591,-48.277,175.061,14.874,152.192
C00614=1094.733,-116.841,-48.267,175.059,14.873,152.192
C00615=1094.728,-117.092,-48.259,175.057,14.872,152.192
C00616=1094.721,-117.341,-48.249,175.055,14.873,152.192
C00617=1094.715,-117.591,-48.239,175.054,14.872,152.193
C00618=1094.709,-117.841,-48.230,175.052,14.872,152.193
C00619=1094.703,-118.091,-48.220,175.050,14.872,152.193
C00620=1094.697,-118.341,-48.211,175.049,14.871,152.194
C00621=1094.691,-118.590,-48.201,175.047,14.871,152.194
C00622=1094.684,-118.840,-48.192,175.046,14.871,152.194
C00623=1094.679,-119.089,-48.182,175.044,14.870,152.195
C00624=1094.672,-119.339,-48.173,175.043,14.871,152.195
C00625=1094.666,-119.589,-48.164,175.041,14.870,152.195
C00626=1094.660,-119.838,-48.154,175.038,14.870,152.196
C00627=1094.653,-120.088,-48.145,175.037,14.870,152.196
C00628=1094.647,-120.339,-48.136,175.035,14.869,152.196
C00629=1094.641,-120.588,-48.126,175.034,14.870,152.197
C00630=1094.635,-120.838,-48.117,175.032,14.869,152.197
C00631=1094.630,-121.087,-48.108,175.031,14.869,152.197
C00632=1094.623,-121.337,-48.098,175.029,14.869,152.197
C00633=1094.616,-121.587,-48.089,175.028,14.868,152.198
C00634=1094.610,-121.836,-48.079,175.025,14.868,152.198
C00635=1094.604,-122.086,-48.070,175.024,14.868,152.198
C00636=1094.598,-122.337,-48.061,175.022,14.868,152.199
C00637=1094.592,-122.586,-48.052,175.021,14.868,152.199
C00638=1094.587,-122.835,-48.042,175.019,14.867,152.199
C00639=1094.580,-123.085,-48.033,175.018,14.868,152.200
C00640=1094.573,-123.335,-48.024,175.016,14.867,152.200
C00641=1094.567,-123.585,-48.014,175.014,14.867,152.200
C00642=1094.561,-123.835,-48.005,175.013,14.867,152.201
C00643=1094.555,-124.085,-47.996,175.011,14.867,152.201
C00644=1094.549,-124.335,-47.986,175.009,14.866,152.201
C00645=1094.544,-124.584,-47.977,175.008,14.866,152.201
C00646=1094.537,-124.833,-47.968,175.006,14.866,152.202
C00647=1094.531,-125.084,-47.959,175.005,14.866,152.202
C00648=1094.525,-125.333,-47.950,175.003,14.866,152.203
C00649=1094.518,-125.583,-47.940,175.001,14.866,152.203
C00650=1094.511,-125.833,-47.931,174.999,14.865,152.203
C00651=1094.506,-126.082,-47.923,174.998,14.865,152.203
C00652=1094.500,-126.332,-47.913,174.996,14.865,152.204
C00653=1094.494,-126.582,-47.903,174.995,14.865,152.204
C00654=1094.487,-126.831,-47.894,174.993,14.865,152.205
C00655=1094.481,-127.082,-47.886,174.992,14.865,152.205
C00656=1094.475,-127.332,-47.876,174.989,14.864,152.205
C00657=1094.468,-127.593,-47.867,174.987,14.864,152.205
C00658=1094.462,-127.852,-47.857,174.986,14.864,152.206
C00659=1094.456,-128.114,-47.847,174.984,14.863,152.206
C00660=1094.457,-128.373,-47.835,174.983,14.861,152.206
C00661=1094.050,-128.393,-47.948,174.938,14.970,152.237
C00662=1094.047,-128.135,-47.961,174.939,14.972,152.237
C00663=1094.054,-127.874,-47.970,174.941,14.973,152.237
C00664=1094.060,-127.614,-47.979,174.942,14.973,152.236
C00665=1094.067,-127.354,-47.989,174.944,14.973,152.236
C00666=1094.072,-127.103,-47.998,174.947,14.974,152.235
C00667=1094.079,-126.854,-48.007,174.948,14.974,152.235
C00668=1094.086,-126.604,-48.016,174.950,14.974,152.235
C00669=1094.092,-126.354,-48.026,174.951,14.974,152.235
C00670=1094.097,-126.105,-48.034,174.953,14.975,152.234
C00671=1094.104,-125.855,-48.043,174.954,14.974,152.234
C00672=1094.110,-125.605,-48.053,174.956,14.975,152.234
C00673=1094.116,-125.356,-48.062,174.958,14.975,152.233
C00674=1094.122,-125.106,-48.072,174.959,14.975,152.233
C00675=1094.129,-124.856,-48.080,174.961,14.975,152.233
C00676=1094.135,-124.607,-48.090,174.963,14.975,152.232
C00677=1094.141,-124.357,-48.099,174.964,14.976,152.232
C00678=1094.147,-124.107,-48.109,174.966,14.976,152.232
C00679=1094.153,-123.856,-48.118,174.967,14.976,152.231
C00680=1094.159,-123.607,-48.127,174.969,14.976,152.231
C00681=1094.166,-123.357,-48.136,174.971,14.976,152.231
C00682=1094.171,-123.108,-48.145,174.972,14.977,152.231
C00683=1094.178,-122.858,-48.155,174.974,14.976,152.230
C00684=1094.184,-122.609,-48.164,174.976,14.977,152.230
C00685=1094.190,-122.358,-48.173,174.977,14.977,152.230
C00686=1094.196,-122.108,-48.183,174.979,14.977,152.229
C00687=1094.202,-121.859,-48.192,174.980,14.978,152.229
C00688=1094.209,-121.609,-48.201,174.982,14.978,152.229
C00689=1094.214,-121.360,-48.211,174.983,14.978,152.228
C00690=1094.221,-121.110,-48.220,174.985,14.978,152.228
C00691=1094.227,-120.860,-48.230,174.988,14.979,152.228
C00692=1094.233,-120.610,-48.239,174.989,14.979,152.227
C00693=1094.239,-120.360,-48.248,174.991,14.979,152.227
C00694=1094.245,-120.110,-48.258,174.992,14.979,152.227
C00695=1094.251,-119.861,-48.267,174.994,14.980,152.226
C00696=1094.258,-119.611,-48.276,174.995,14.980,152.226
C00697=1094.264,-119.362,-48.285,174.997,14.980,152.226
C00698=1094.270,-119.112,-48.295,174.998,14.980,152.226
C00699=1094.276,-118.862,-48.305,175.001,14.980,152.225
C00700=1094.282,-118.613,-48.314,175.002,14.980,152.225
C00701=1094.288,-118.363,-48.324,175.004,14.981,152.225
C00702=1094.294,-118.112,-48.333,175.006,14.981,152.224
C00703=1094.300,-117.863,-48.342,175.007,14.981,152.224
C00704=1094.307,-117.613,-48.352,175.009,14.982,152.224
C00705=1094.313,-117.363,-48.361,175.010,14.982,152.224
C00706=1094.318,-117.114,-48.370,175.012,14.982,152.223
C00707=1094.324,-116.864,-48.380,175.013,14.983,152.223
C00708=1094.331,-116.614,-48.390,175.015,14.983,152.223
C00709=1094.337,-116.364,-48.399,175.016,14.983,152.222
C00710=1094.343,-116.115,-48.409,175.018,14.983,152.222
C00711=1094.350,-115.865,-48.418,175.020,14.984,152.222
C00712=1094.356,-115.615,-48.427,175.022,14.984,152.221
C00713=1094.362,-115.366,-48.437,175.024,14.984,152.221
C00714=1094.368,-115.116,-48.446,175.025,14.985,152.221
C00715=1094.375,-114.866,-48.456,175.027,14.985,152.220
C00716=1094.381,-114.616,-48.465,175.028,14.985,152.220
C00717=1094.387,-114.366,-48.475,175.030,14.986,152.220
C00718=1094.393,-114.117,-48.485,175.032,14.986,152.220
C00719=1094.399,-113.867,-48.494,175.033,14.986,152.219
C00720=1094.404,-113.617,-48.504,175.035,14.987,152.219
C00721=1094.410,-113.368,-48.514,175.036,14.987,152.219
C00722=1094.417,-113.102,-48.524,175.038,14.987,152.218
C00723=1094.423,-112.837,-48.534,175.040,14.988,152.218
C00724=1094.430,-112.572,-48.544,175.041,14.988,152.218
C00725=1094.437,-112.307,-48.555,175.043,14.988,152.218
C00726=1094.443,-112.057,-48.564,175.046,14.989,152.217
C00727=1094.449,-111.807,-48.574,175.047,14.989,152.217
C00728=1094.455,-111.557,-48.584,175.049,14.989,152.217
C00729=1094.461,-111.308,-48.593,175.050,14.989,152.216
C00730=1094.468,-111.058,-48.603,175.052,14.990,152.216
C00731=1094.474,-110.808,-48.612,175.054,14.990,152.216
C00732=1094.479,-110.559,-48.621,175.055,14.990,152.215
C00733=1094.485,-110.309,-48.631,175.057,14.991,152.215
C00734=1094.492,-110.060,-48.641,175.058,14.991,152.215
C00735=1094.498,-109.810,-48.651,175.060,14.991,152.215
C00736=1094.504,-109.560,-48.660,175.062,14.992,152.214
C00737=1094.510,-109.310,-48.671,175.063,14.992,152.214
C00738=1094.516,-109.060,-48.680,175.065,14.992,152.214
C00739=1094.522,-108.811,-48.690,175.066,14.992,152.213
C00740=1094.528,-108.561,-48.699,175.068,14.993,152.213
C00741=1094.535,-108.312,-48.710,175.070,14.994,152.213
C00742=1094.541,-108.062,-48.719,175.071,14.994,152.213
C00743=1094.547,-107.812,-48.729,175.073,14.994,152.212
C00744=1094.553,-107.562,-48.738,175.075,14.995,152.212
C00745=1094.559,-107.312,-48.748,175.076,14.995,152.212
C00746=1094.565,-107.062,-48.758,175.078,14.996,152.211
C00747=1094.571,-106.813,-48.768,175.079,14.996,152.211
C00748=1094.577,-106.563,-48.778,175.082,14.996,152.211
C00749=1094.584,-106.314,-48.787,175.084,14.997,152.211
C00750=1094.589,-106.063,-48.798,175.085,14.997,152.210
C00751=1094.595,-105.814,-48.807,175.087,14.997,152.210
C00752=1094.602,-105.564,-48.817,175.088,14.998,152.210
C00753=1094.608,-105.315,-48.827,175.090,14.998,152.210
C00754=1094.614,-105.065,-48.837,175.091,14.999,152.209
C00755=1094.619,-104.815,-48.847,175.093,14.999,152.209
C00756=1094.626,-104.565,-48.856,175.095,14.999,152.209
C00757=1094.632,-104.316,-48.867,175.097,15.000,152.208
C00758=1094.638,-104.066,-48.876,175.098,15.000,152.208
C00759=1094.644,-103.816,-48.886,175.100,15.001,152.208
C00760=1094.650,-103.566,-48.896,175.102,15.001,152.208
C00761=1094.656,-103.317,-48.906,175.103,15.001,152.207
C00762=1094.663,-103.067,-48.916,175.105,15.002,152.207
C00763=1094.668,-102.817,-48.926,175.107,15.002,152.207
C00764=1094.674,-102.568,-48.936,175.108,15.003,152.206
C00765=1094.681,-102.318,-48.946,175.110,15.003,152.206
C00766=1094.687,-102.068,-48.955,175.111,15.003,152.206
C00767=1094.692,-101.818,-48.965,175.113,15.004,152.206
C00768=1094.699,-101.569,-48.976,175.115,15.005,152.205
C00769=1094.705,-101.319,-48.985,175.116,15.004,152.205
C00770=1094.710,-101.069,-48.995,175.118,15.005,152.205
C00771=1094.717,-100.819,-49.006,175.120,15.006,152.204
C00772=1094.724,-100.569,-49.016,175.121,15.006,152.204
C00773=1094.730,-100.320,-49.025,175.123,15.007,152.204
C00774=1094.735,-100.070,-49.036,175.125,15.007,152.204
C00775=1094.742,-99.820,-49.046,175.126,15.007,152.204
C00776=1094.748,-99.570,-49.055,175.128,15.008,152.203
C00777=1094.754,-99.321,-49.066,175.130,15.008,152.203
C00778=1094.760,-99.071,-49.076,175.131,15.008,152.203
C00779=1094.766,-98.821,-49.085,175.133,15.009,152.202
C00780=1094.772,-98.572,-49.096,175.135,15.010,152.202
C00781=1094.778,-98.322,-49.106,175.136,15.010,152.202
C00782=1094.784,-98.073,-49.116,175.138,15.011,152.202
C00783=1094.790,-97.823,-49.126,175.140,15.011,152.201
C00784=1094.796,-97.573,-49.136,175.141,15.011,152.201
C00785=1094.802,-97.324,-49.146,175.143,15.012,152.201
C00786=1094.809,-97.049,-49.158,175.145,15.013,152.201
C00787=1094.816,-96.775,-49.169,175.147,15.013,152.200
C00788=1094.822,-96.501,-49.180,175.149,15.014,152.200
C00789=1094.828,-96.227,-49.191,175.151,15.014,152.200
C00790=1094.835,-95.977,-49.201,175.152,15.014,152.199
C00791=1094.840,-95.727,-49.211,175.154,15.015,152.199
C00792=1094.847,-95.478,-49.221,175.155,15.016,152.199
C00793=1094.852,-95.228,-49.231,175.157,15.016,152.199
C00794=1094.858,-94.978,-49.242,175.158,15.017,152.198
C00795=1094.864,-94.728,-49.252,175.160,15.017,152.198
C00796=1094.870,-94.479,-49.262,175.161,15.017,152.198
C00797=1094.876,-94.228,-49.273,175.163,15.018,152.198
C00798=1094.883,-93.979,-49.283,175.165,15.019,152.197
C00799=1094.888,-93.729,-49.293,175.167,15.020,152.197
C00800=1094.895,-93.480,-49.303,175.168,15.020,152.197
C00801=1094.900,-93.230,-49.314,175.170,15.020,152.197
C00802=1094.907,-92.981,-49.324,175.172,15.021,152.196
C00803=1094.912,-92.730,-49.334,175.173,15.021,152.196
C00804=1094.919,-92.481,-49.344,175.175,15.022,152.196
C00805=1094.924,-92.231,-49.354,175.177,15.023,152.196
C00806=1094.931,-91.982,-49.365,175.178,15.023,152.195
C00807=1094.936,-91.732,-49.375,175.180,15.023,152.195
C00808=1094.943,-91.482,-49.386,175.182,15.024,152.195
C00809=1094.948,-91.232,-49.396,175.184,15.025,152.194
C00810=1094.955,-90.983,-49.406,175.185,15.025,152.194
C00811=1094.960,-90.733,-49.416,175.187,15.026,152.194
C00812=1094.966,-90.483,-49.427,175.189,15.026,152.194
C00813=1094.973,-90.234,-49.437,175.190,15.027,152.193
C00814=1094.978,-89.984,-49.447,175.192,15.027,152.193
C00815=1094.985,-89.735,-49.458,175.193,15.028,152.193
C00816=1094.991,-89.484,-49.468,175.195,15.028,152.193
C00817=1094.997,-89.235,-49.479,175.196,15.029,152.192
C00818=1095.003,-88.985,-49.489,175.198,15.029,152.192
C00819=1095.009,-88.735,-49.499,175.200,15.030,152.192
C00820=1095.015,-88.486,-49.510,175.202,15.031,152.192
C00821=1095.020,-88.236,-49.520,175.203,15.031,152.191
C00822=1095.027,-87.986,-49.531,175.205,15.031,152.191
C00823=1095.033,-87.736,-49.542,175.207,15.032,152.191
C00824=1095.039,-87.487,-49.551,175.209,15.033,152.191
C00825=1095.045,-87.237,-49.562,175.210,15.033,152.190
C00826=1095.051,-86.988,-49.572,175.212,15.034,152.190
C00827=1095.057,-86.738,-49.582,175.214,15.034,152.190
C00828=1095.063,-86.488,-49.594,175.216,15.035,152.190
C00829=1095.070,-86.238,-49.604,175.217,15.035,152.189
C00830=1095.075,-85.988,-49.614,175.219,15.036,152.189
C00831=1095.081,-85.739,-49.624,175.221,15.037,152.189
C00832=1095.087,-85.490,-49.635,175.222,15.037,152.189
C00833=1095.093,-85.239,-49.646,175.224,15.037,152.188
C00834=1095.100,-84.990,-49.656,175.225,15.038,152.188
C00835=1095.105,-84.740,-49.667,175.227,15.039,152.188
C00836=1095.111,-84.490,-49.677,175.229,15.039,152.188
C00837=1095.118,-84.240,-49.688,175.230,15.040,152.187
C00838=1095.124,-83.991,-49.699,175.232,15.040,152.187
C00839=1095.130,-83.742,-49.709,175.234,15.041,152.187
C00840=1095.136,-83.491,-49.719,175.236,15.042,152.187
C00841=1095.141,-83.242,-49.730,175.237,15.042,152.187
C00842=1095.148,-82.992,-49.741,175.239,15.043,152.186
C00843=1095.154,-82.743,-49.752,175.241,15.044,152.186
C00844=1095.160,-82.492,-49.762,175.242,15.044,152.186
C00845=1095.166,-82.243,-49.772,175.244,15.044,152.185
C00846=1095.172,-81.993,-49.783,175.245,15.045,152.185
C00847=1095.179,-81.744,-49.793,175.247,15.046,152.185
C00848=1095.184,-81.494,-49.804,175.249,15.047,152.185
C00849=1095.191,-81.244,-49.815,175.250,15.047,152.184
C00850=1095.197,-80.972,-49.826,175.252,15.047,152.184
C00851=1095.204,-80.701,-49.838,175.254,15.048,152.184
C00852=1095.211,-80.428,-49.849,175.256,15.049,152.184
C00853=1095.218,-80.156,-49.861,175.258,15.049,152.183
C00854=1095.223,-79.907,-49.872,175.260,15.050,152.183
C00855=1095.229,-79.657,-49.883,175.262,15.051,152.183
C00856=1095.235,-79.408,-49.893,175.264,15.052,152.183
C00857=1095.241,-79.158,-49.903,175.265,15.052,152.182
C00858=1095.247,-78.908,-49.915,175.267,15.052,152.182
C00859=1095.253,-78.658,-49.925,175.268,15.053,152.182
C00860=1095.259,-78.409,-49.936,175.270,15.054,152.182
C00861=1095.264,-78.159,-49.947,175.271,15.054,152.182
C00862=1095.272,-77.909,-49.958,175.273,15.055,152.181
C00863=1095.277,-77.660,-49.969,175.275,15.056,152.181
C00864=1095.283,-77.410,-49.980,175.277,15.057,152.181
C00865=1095.288,-77.160,-49.990,175.279,15.057,152.180
C00866=1095.295,-76.910,-50.001,175.280,15.057,152.180
C00867=1095.301,-76.661,-50.012,175.282,15.058,152.180
C00868=1095.307,-76.411,-50.022,175.284,15.059,152.180
C00869=1095.313,-76.162,-50.033,175.285,15.060,152.180
C00870=1095.319,-75.912,-50.044,175.287,15.061,152.179
C00871=1095.325,-75.662,-50.055,175.289,15.061,152.179
C00872=1095.331,-75.413,-50.066,175.290,15.061,152.179
C00873=1095.337,-75.163,-50.077,175.292,15.062,152.179
C00874=1095.343,-74.913,-50.088,175.294,15.063,152.178
C00875=1095.349,-74.664,-50.098,175.296,15.064,152.178
C00876=1095.355,-74.414,-50.110,175.298,15.064,152.178
C00877=1095.361,-74.164,-50.121,175.298,15.065,152.178
C00878=1095.367,-73.914,-50.131,175.300,15.066,152.177
C00879=1095.372,-73.665,-50.142,175.302,15.066,152.177
C00880=1095.379,-73.414,-50.153,175.304,15.067,152.177
C00881=1095.384,-73.165,-50.164,175.306,15.068,152.177
C00882=1095.390,-72.915,-50.175,175.307,15.069,152.177
C00883=1095.396,-72.666,-50.185,175.309,15.069,152.176
C00884=1095.402,-72.416,-50.197,175.310,15.070,152.176
C00885=1095.408,-72.166,-50.208,175.312,15.070,152.176
C00886=1095.414,-71.917,-50.218,175.314,15.071,152.176
C00887=1095.420,-71.667,-50.229,175.316,15.072,152.175
C00888=1095.426,-71.417,-50.241,175.318,15.073,152.175
C00889=1095.431,-71.167,-50.252,175.319,15.073,152.175
C00890=1095.437,-70.918,-50.263,175.321,15.074,152.175
C00891=1095.442,-70.668,-50.274,175.323,15.074,152.174
C00892=1095.449,-70.419,-50.286,175.324,15.076,152.174
C00893=1095.455,-70.169,-50.297,175.326,15.076,152.174
C00894=1095.460,-69.920,-50.308,175.328,15.077,152.174
C00895=1095.467,-69.670,-50.319,175.329,15.077,152.174
C00896=1095.473,-69.420,-50.330,175.331,15.078,152.173
C00897=1095.478,-69.171,-50.341,175.332,15.079,152.173
C00898=1095.485,-68.920,-50.352,175.334,15.080,152.173
C00899=1095.490,-68.671,-50.363,175.336,15.081,152.173
C00900=1095.496,-68.421,-50.374,175.338,15.081,152.172
C00901=1095.502,-68.172,-50.384,175.340,15.082,152.172
C00902=1095.508,-67.922,-50.396,175.341,15.083,152.172
C00903=1095.513,-67.672,-50.407,175.343,15.083,152.172
C00904=1095.519,-67.423,-50.419,175.345,15.084,152.172
C00905=1095.526,-67.173,-50.430,175.346,15.085,152.171
C00906=1095.531,-66.923,-50.441,175.348,15.086,152.171
C00907=1095.538,-66.673,-50.452,175.350,15.087,152.171
C00908=1095.543,-66.424,-50.463,175.352,15.087,152.171
C00909=1095.549,-66.174,-50.474,175.354,15.088,152.170
C00910=1095.555,-65.924,-50.485,175.354,15.089,152.170
C00911=1095.562,-65.675,-50.497,175.356,15.089,152.170
C00912=1095.567,-65.425,-50.508,175.358,15.090,152.170
C00913=1095.573,-65.175,-50.519,175.360,15.091,152.170
C00914=1095.579,-64.906,-50.531,175.362,15.091,152.169
C00915=1095.586,-64.636,-50.543,175.364,15.093,152.169
C00916=1095.591,-64.366,-50.555,175.366,15.093,152.169
C00917=1095.599,-64.097,-50.568,175.367,15.094,152.169
C00918=1095.605,-63.847,-50.579,175.369,15.095,152.168
C00919=1095.610,-63.597,-50.591,175.371,15.095,152.168
C00920=1095.616,-63.347,-50.601,175.373,15.096,152.168
C00921=1095.622,-63.098,-50.613,175.375,15.097,152.168
C00922=1095.628,-62.848,-50.624,175.376,15.097,152.168
C00923=1095.634,-62.599,-50.635,175.378,15.098,152.167
C00924=1095.641,-62.349,-50.646,175.380,15.099,152.167
C00925=1095.646,-62.099,-50.659,175.381,15.100,152.167
C00926=1095.652,-61.850,-50.669,175.383,15.101,152.167
C00927=1095.658,-61.600,-50.681,175.385,15.101,152.166
C00928=1095.664,-61.351,-50.692,175.387,15.102,152.166
C00929=1095.670,-61.101,-50.704,175.389,15.103,152.166
C00930=1095.676,-60.851,-50.714,175.390,15.104,152.166
C00931=1095.682,-60.601,-50.726,175.392,15.105,152.166
C00932=1095.688,-60.352,-50.738,175.393,15.105,152.165
C00933=1095.693,-60.102,-50.749,175.395,15.106,152.165
C00934=1095.700,-59.852,-50.760,175.397,15.106,152.165
C00935=1095.706,-59.603,-50.772,175.399,15.107,152.165
C00936=1095.711,-59.353,-50.783,175.400,15.108,152.164
C00937=1095.717,-59.103,-50.794,175.402,15.109,152.164
C00938=1095.724,-58.854,-50.806,175.404,15.110,152.164
C00939=1095.730,-58.604,-50.817,175.406,15.111,152.164
C00940=1095.736,-58.354,-50.828,175.408,15.112,152.164
C00941=1095.741,-58.105,-50.841,175.410,15.112,152.163
C00942=1095.748,-57.855,-50.852,175.411,15.112,152.163
C00943=1095.754,-57.606,-50.863,175.413,15.113,152.163
C00944=1095.760,-57.355,-50.875,175.414,15.114,152.163
C00945=1095.766,-57.106,-50.885,175.416,15.115,152.162
C00946=1095.772,-56.856,-50.898,175.418,15.116,152.162
C00947=1095.777,-56.607,-50.909,175.420,15.116,152.162
C00948=1095.784,-56.357,-50.921,175.422,15.117,152.162
C00949=1095.790,-56.108,-50.932,175.423,15.118,152.162
C00950=1095.796,-55.858,-50.944,175.425,15.119,152.161
C00951=1095.801,-55.608,-50.955,175.427,15.120,152.161
C00952=1095.808,-55.358,-50.966,175.429,15.120,152.161
C00953=1095.814,-55.109,-50.978,175.431,15.121,152.160
C00954=1095.819,-54.859,-50.990,175.432,15.122,152.160
C00955=1095.825,-54.610,-51.001,175.433,15.122,152.160
C00956=1095.832,-54.360,-51.013,175.435,15.123,152.160
C00957=1095.838,-54.110,-51.025,175.437,15.124,152.160
C00958=1095.843,-53.860,-51.036,175.439,15.125,152.160
C00959=1095.850,-53.611,-51.048,175.441,15.126,152.159
C00960=1095.856,-53.361,-51.059,175.443,15.126,152.159
C00961=1095.862,-53.111,-51.072,175.444,15.127,152.159
C00962=1095.867,-52.862,-51.082,175.446,15.128,152.158
C00963=1095.874,-52.612,-51.094,175.448,15.129,152.158
C00964=1095.880,-52.362,-51.106,175.450,15.130,152.158
C00965=1095.886,-52.113,-51.118,175.452,15.130,152.158
C00966=1095.892,-51.863,-51.130,175.454,15.131,152.158
C00967=1095.898,-51.614,-51.141,175.455,15.132,152.157
C00968=1095.904,-51.364,-51.153,175.456,15.133,152.157
C00969=1095.910,-51.114,-51.164,175.458,15.133,152.157
C00970=1095.916,-50.865,-51.176,175.460,15.134,152.157
C00971=1095.922,-50.614,-51.188,175.462,15.135,152.156
C00972=1095.928,-50.365,-51.199,175.464,15.135,152.156
C00973=1095.934,-50.116,-51.212,175.465,15.137,152.156
C00974=1095.940,-49.866,-51.223,175.467,15.137,152.156
C00975=1095.946,-49.616,-51.235,175.469,15.138,152.156
C00976=1095.951,-49.367,-51.246,175.471,15.139,152.155
C00977=1095.957,-49.117,-51.259,175.473,15.140,152.155
C00978=1095.964,-48.849,-51.271,175.475,15.141,152.155
C00979=1095.970,-48.580,-51.284,175.476,15.141,152.155
C00980=1095.976,-48.312,-51.297,175.478,15.142,152.155
C00981=1095.983,-48.043,-51.309,175.481,15.144,152.154
C00982=1095.988,-47.794,-51.321,175.482,15.144,152.154
C00983=1095.995,-47.544,-51.333,175.484,15.145,152.154
C00984=1096.000,-47.294,-51.345,175.485,15.146,152.154
C00985=1096.006,-47.045,-51.357,175.487,15.147,152.153
C00986=1096.012,-46.795,-51.369,175.489,15.147,152.153
C00987=1096.017,-46.545,-51.381,175.491,15.148,152.153
C00988=1096.024,-46.296,-51.393,175.492,15.149,152.153
C00989=1096.029,-46.046,-51.405,175.494,15.150,152.153
C00990=1096.036,-45.796,-51.416,175.496,15.151,152.152
C00991=1096.041,-45.547,-51.428,175.498,15.152,152.152
C00992=1096.048,-45.298,-51.440,175.500,15.152,152.152
C00993=1096.053,-45.048,-51.453,175.502,15.153,152.152
C00994=1096.058,-44.798,-51.464,175.503,15.154,152.152
C00995=1096.065,-44.548,-51.476,175.505,15.155,152.151
C00996=1096.070,-44.299,-51.488,175.507,15.156,152.151
C00997=1096.077,-44.049,-51.500,175.508,15.157,152.151
C00998=1096.083,-43.799,-51.512,175.510,15.158,152.151
C00999=1096.089,-43.550,-51.524,175.512,15.158,152.150
C01000=1096.095,-43.300,-51.536,175.514,15.159,152.150
C01001=1096.101,-43.050,-51.549,175.516,15.160,152.150
C01002=1096.106,-42.801,-51.560,175.518,15.161,152.150
C01003=1096.112,-42.551,-51.572,175.519,15.162,152.150
C01004=1096.118,-42.302,-51.584,175.521,15.162,152.149
C01005=1096.124,-42.052,-51.596,175.523,15.164,152.149
C01006=1096.130,-41.802,-51.608,175.525,15.164,152.149
C01007=1096.136,-41.553,-51.620,175.527,15.165,152.149
C01008=1096.142,-41.303,-51.632,175.528,15.166,152.149
C01009=1096.148,-41.053,-51.645,175.530,15.167,152.148
C01010=1096.154,-40.804,-51.657,175.532,15.168,152.148
C01011=1096.160,-40.554,-51.669,175.534,15.168,152.148
C01012=1096.166,-40.304,-51.680,175.536,15.170,152.148
C01013=1096.171,-40.055,-51.693,175.537,15.170,152.147
C01014=1096.177,-39.805,-51.705,175.539,15.171,152.147
C01015=1096.184,-39.556,-51.717,175.541,15.172,152.147
C01016=1096.190,-39.306,-51.730,175.543,15.173,152.147
C01017=1096.195,-39.056,-51.742,175.545,15.174,152.147
C01018=1096.202,-38.807,-51.754,175.547,15.174,152.146
C01019=1096.208,-38.557,-51.766,175.548,15.175,152.146
C01020=1096.213,-38.308,-51.779,175.550,15.176,152.146
C01021=1096.218,-38.057,-51.790,175.552,15.177,152.146
C01022=1096.224,-37.807,-51.803,175.554,15.178,152.145
C01023=1096.230,-37.559,-51.815,175.555,15.179,152.145
C01024=1096.236,-37.309,-51.827,175.557,15.180,152.145
C01025=1096.242,-37.059,-51.839,175.559,15.180,152.145
C01026=1096.247,-36.810,-51.852,175.561,15.182,152.145
C01027=1096.253,-36.560,-51.864,175.563,15.182,152.144
C01028=1096.260,-36.310,-51.876,175.564,15.183,152.144
C01029=1096.265,-36.061,-51.889,175.566,15.184,152.144
C01030=1096.271,-35.811,-51.901,175.568,15.185,152.144
C01031=1096.277,-35.561,-51.914,175.570,15.186,152.144
C01032=1096.282,-35.312,-51.926,175.571,15.187,152.143
C01033=1096.288,-35.062,-51.938,175.573,15.188,152.143
C01034=1096.295,-34.813,-51.950,175.575,15.188,152.143
C01035=1096.300,-34.563,-51.963,175.578,15.190,152.143
C01036=1096.306,-34.314,-51.975,175.579,15.191,152.143
C01037=1096.312,-34.064,-51.988,175.581,15.191,152.142
C01038=1096.318,-33.814,-52.000,175.583,15.192,152.142
C01039=1096.323,-33.565,-52.012,175.585,15.193,152.142
C01040=1096.330,-33.315,-52.024,175.587,15.194,152.142
C01041=1096.336,-33.065,-52.037,175.588,15.195,152.141
C01042=1096.342,-32.797,-52.050,175.590,15.196,152.141
C01043=1096.349,-32.529,-52.064,175.592,15.197,152.141
C01044=1096.354,-32.261,-52.077,175.594,15.197,152.141
C01045=1096.361,-31.993,-52.090,175.597,15.199,152.140
C01046=1096.366,-31.743,-52.103,175.598,15.199,152.140
C01047=1096.372,-31.493,-52.115,175.600,15.201,152.140
C01048=1096.378,-31.244,-52.128,175.602,15.201,152.140
C01049=1096.384,-30.994,-52.140,175.604,15.202,152.140
C01050=1096.390,-30.745,-52.153,175.605,15.203,152.139
C01051=1096.396,-30.496,-52.165,175.607,15.204,152.139
C01052=1096.402,-30.246,-52.178,175.609,15.205,152.139
C01053=1096.408,-29.996,-52.190,175.611,15.205,152.139
C01054=1096.413,-29.747,-52.202,175.613,15.207,152.139
C01055=1096.419,-29.497,-52.215,175.614,15.207,152.138
C01056=1096.425,-29.247,-52.228,175.616,15.208,152.138
C01057=1096.431,-28.998,-52.241,175.618,15.209,152.138
C01058=1096.437,-28.748,-52.253,175.620,15.210,152.138
C01059=1096.443,-28.499,-52.266,175.622,15.211,152.137
C01060=1096.449,-28.249,-52.278,175.624,15.211,152.137
C01061=1096.455,-27.999,-52.290,175.625,15.213,152.137
C01062=1096.461,-27.750,-52.303,175.627,15.213,152.137
C01063=1096.467,-27.500,-52.316,175.629,15.214,152.137
C01064=1096.473,-27.250,-52.328,175.632,15.215,152.136
C01065=1096.478,-27.001,-52.341,175.633,15.217,152.136
C01066=1096.484,-26.751,-52.353,175.635,15.217,152.136
C01067=1096.491,-26.502,-52.366,175.637,15.218,152.136
C01068=1096.497,-26.252,-52.379,175.639,15.219,152.135
C01069=1096.502,-26.002,-52.392,175.640,15.220,152.135
C01070=1096.507,-25.752,-52.404,175.642,15.221,152.135
C01071=1096.513,-25.503,-52.418,175.644,15.221,152.135
C01072=1096.519,-25.253,-52.430,175.646,15.223,152.135
C01073=1096.525,-25.003,-52.443,175.648,15.223,152.134
C01074=1096.531,-24.754,-52.455,175.649,15.224,152.134
C01075=1096.537,-24.505,-52.468,175.651,15.225,152.134
C01076=1096.542,-24.255,-52.481,175.653,15.226,152.134
C01077=1096.548,-24.005,-52.493,175.656,15.227,152.134
C01078=1096.555,-23.756,-52.507,175.657,15.228,152.133
C01079=1096.560,-23.506,-52.520,175.659,15.229,152.133
C01080=1096.565,-23.257,-52.532,175.661,15.230,152.133
C01081=1096.571,-23.007,-52.544,175.663,15.231,152.133
C01082=1096.577,-22.757,-52.558,175.664,15.232,152.133
C01083=1096.583,-22.508,-52.570,175.666,15.232,152.132
C01084=1096.589,-22.258,-52.584,175.668,15.233,152.132
C01085=1096.595,-22.008,-52.596,175.670,15.234,152.132
C01086=1096.601,-21.759,-52.609,175.672,15.235,152.132
C01087=1096.606,-21.510,-52.622,175.673,15.236,152.131
C01088=1096.612,-21.260,-52.635,175.676,15.237,152.131
C01089=1096.618,-21.010,-52.647,175.678,15.238,152.131
C01090=1096.624,-20.761,-52.661,175.680,15.239,152.131
C01091=1096.630,-20.511,-52.673,175.682,15.240,152.131
C01092=1096.636,-20.261,-52.686,175.683,15.240,152.130
C01093=1096.641,-20.011,-52.699,175.685,15.242,152.130
C01094=1096.647,-19.761,-52.712,175.687,15.242,152.130
C01095=1096.653,-19.513,-52.725,175.689,15.243,152.130
C01096=1096.659,-19.263,-52.737,175.691,15.244,152.129
C01097=1096.665,-19.014,-52.751,175.692,15.245,152.129
C01098=1096.671,-18.764,-52.763,175.695,15.246,152.129
C01099=1096.676,-18.514,-52.777,175.697,15.247,152.129
C01100=1096.682,-18.264,-52.790,175.699,15.248,152.128
C01101=1096.688,-18.015,-52.803,175.700,15.249,152.128
C01102=1096.694,-17.765,-52.816,175.702,15.250,152.128
C01103=1096.701,-17.516,-52.829,175.704,15.250,152.128
C01104=1096.706,-17.266,-52.842,175.706,15.251,152.128
C01105=1096.712,-17.016,-52.855,175.707,15.252,152.128
C01106=1096.718,-16.748,-52.869,175.710,15.254,152.127
C01107=1096.724,-16.479,-52.883,175.712,15.254,152.127
C01108=1096.731,-16.209,-52.897,175.714,15.255,152.127
C01109=1096.737,-15.941,-52.911,175.716,15.256,152.126
C01110=1096.743,-15.691,-52.924,175.718,15.257,152.126
C01111=1096.749,-15.442,-52.937,175.720,15.258,152.126
C01112=1096.755,-15.192,-52.950,175.722,15.259,152.126
C01113=1096.761,-14.943,-52.963,175.724,15.260,152.126
C01114=1096.766,-14.693,-52.977,175.726,15.260,152.125
C01115=1096.772,-14.443,-52.990,175.727,15.262,152.125
C01116=1096.778,-14.194,-53.003,175.729,15.262,152.125
C01117=1096.783,-13.944,-53.016,175.731,15.263,152.125
C01118=1096.789,-13.695,-53.029,175.733,15.265,152.125
C01119=1096.795,-13.445,-53.042,175.735,15.266,152.124
C01120=1096.801,-13.196,-53.055,175.737,15.266,152.124
C01121=1096.807,-12.946,-53.069,175.739,15.267,152.124
C01122=1096.812,-12.696,-53.082,175.741,15.268,152.124
C01123=1096.818,-12.447,-53.095,175.742,15.269,152.123
C01124=1096.824,-12.198,-53.108,175.744,15.270,152.123
C01125=1096.830,-11.947,-53.122,175.747,15.271,152.123
C01126=1096.836,-11.698,-53.135,175.749,15.272,152.123
C01127=1096.841,-11.448,-53.148,175.750,15.273,152.122
C01128=1096.847,-11.199,-53.161,175.752,15.274,152.122
C01129=1096.853,-10.949,-53.175,175.754,15.274,152.122
C01130=1096.859,-10.700,-53.188,175.756,15.276,152.122
C01131=1096.865,-10.450,-53.201,175.758,15.276,152.122
C01132=1096.870,-10.200,-53.215,175.760,15.278,152.121
C01133=1096.876,-9.951,-53.228,175.762,15.278,152.121
C01134=1096.882,-9.701,-53.241,175.764,15.279,152.121
C01135=1096.888,-9.452,-53.254,175.766,15.280,152.121
C01136=1096.894,-9.202,-53.268,175.768,15.281,152.120
C01137=1096.900,-8.953,-53.282,175.769,15.282,152.120
C01138=1096.905,-8.703,-53.294,175.771,15.282,152.120
C01139=1096.911,-8.453,-53.308,175.774,15.284,152.120
C01140=1096.917,-8.204,-53.321,175.776,15.285,152.120
C01141=1096.923,-7.955,-53.335,175.777,15.286,152.119
C01142=1096.929,-7.705,-53.348,175.779,15.286,152.119
C01143=1096.934,-7.455,-53.362,175.781,15.287,152.119
C01144=1096.940,-7.206,-53.375,175.783,15.288,152.119
C01145=1096.946,-6.956,-53.389,175.785,15.289,152.118
C01146=1096.952,-6.706,-53.401,175.787,15.290,152.118
C01147=1096.957,-6.457,-53.415,175.789,15.291,152.118
C01148=1096.964,-6.207,-53.429,175.791,15.292,152.118
C01149=1096.969,-5.957,-53.443,175.793,15.293,152.117
C01150=1096.976,-5.708,-53.456,175.795,15.293,152.117
C01151=1096.981,-5.458,-53.470,175.796,15.294,152.117
C01152=1096.987,-5.209,-53.482,175.799,15.296,152.117
C01153=1096.992,-4.959,-53.496,175.801,15.297,152.116
C01154=1096.999,-4.710,-53.509,175.803,15.297,152.116
C01155=1097.004,-4.460,-53.523,175.805,15.298,152.116
C01156=1097.010,-4.211,-53.537,175.807,15.299,152.116
C01157=1097.016,-3.961,-53.550,175.808,15.300,152.116
C01158=1097.022,-3.712,-53.564,175.811,15.301,152.115
C01159=1097.028,-3.462,-53.578,175.813,15.302,152.115
C01160=1097.034,-3.213,-53.591,175.815,15.303,152.115
C01161=1097.039,-2.962,-53.604,175.817,15.303,152.115
C01162=1097.045,-2.713,-53.618,175.818,15.305,152.114
C01163=1097.051,-2.463,-53.632,175.820,15.305,152.114
C01164=1097.057,-2.214,-53.645,175.823,15.307,152.114
C01165=1097.062,-1.964,-53.659,175.825,15.307,152.114
C01166=1097.068,-1.715,-53.673,175.826,15.308,152.113
C01167=1097.074,-1.465,-53.686,175.828,15.309,152.113
C01168=1097.079,-1.216,-53.700,175.830,15.310,152.113
C01169=1097.085,-0.966,-53.714,175.833,15.311,152.113
C01170=1097.092,-0.696,-53.729,175.834,15.312,152.112
C01171=1097.098,-0.425,-53.744,175.836,15.313,152.112
C01172=1097.103,-0.155,-53.758,175.839,15.314,152.112
C01173=1097.110,0.116,-53.773,175.841,15.315,152.112
C01174=1097.116,0.365,-53.787,175.842,15.316,152.112
C01175=1097.121,0.615,-53.801,175.844,15.317,152.111
C01176=1097.127,0.864,-53.815,175.847,15.318,152.111
C01177=1097.133,1.114,-53.828,175.849,15.319,152.111
C01178=1097.138,1.363,-53.842,175.851,15.319,152.111
C01179=1097.144,1.614,-53.856,175.852,15.321,152.110
C01180=1097.150,1.863,-53.870,175.854,15.321,152.110
C01181=1097.156,2.112,-53.884,175.857,15.323,152.110
C01182=1097.162,2.361,-53.898,175.859,15.323,152.110
C01183=1097.167,2.611,-53.912,175.861,15.324,152.109
C01184=1097.173,2.861,-53.925,175.863,15.325,152.109
C01185=1097.178,3.110,-53.939,175.864,15.326,152.109
C01186=1097.185,3.360,-53.953,175.867,15.327,152.109
C01187=1097.191,3.610,-53.967,175.869,15.328,152.108
C01188=1097.196,3.859,-53.981,175.871,15.329,152.108
C01189=1097.201,4.109,-53.995,175.872,15.330,152.108
C01190=1097.207,4.358,-54.008,175.874,15.330,152.108
C01191=1097.213,4.607,-54.022,175.877,15.332,152.107
C01192=1097.220,4.857,-54.037,175.879,15.332,152.107
C01193=1097.225,5.107,-54.051,175.881,15.333,152.107
C01194=1097.230,5.356,-54.064,175.882,15.334,152.107
C01195=1097.236,5.606,-54.078,175.884,15.335,152.107
C01196=1097.242,5.855,-54.092,175.887,15.336,152.106
C01197=1097.249,6.105,-54.106,175.889,15.337,152.106
C01198=1097.254,6.355,-54.120,175.891,15.338,152.106
C01199=1097.260,6.604,-54.134,175.893,15.338,152.105
C01200=1097.265,6.854,-54.148,175.894,15.339,152.105
C01201=1097.270,7.103,-54.162,175.897,15.341,152.105
C01202=1097.278,7.353,-54.176,175.899,15.341,152.105
C01203=1097.283,7.602,-54.190,175.901,15.342,152.104
C01204=1097.289,7.852,-54.204,175.903,15.343,152.104
C01205=1097.294,8.101,-54.218,175.905,15.344,152.104
C01206=1097.300,8.351,-54.233,175.907,15.345,152.104
C01207=1097.306,8.601,-54.247,175.909,15.346,152.104
C01208=1097.311,8.850,-54.261,175.911,15.347,152.103
C01209=1097.317,9.100,-54.274,175.913,15.347,152.103
C01210=1097.324,9.349,-54.289,175.915,15.349,152.103
C01211=1097.329,9.599,-54.303,175.917,15.349,152.102
C01212=1097.335,9.848,-54.316,175.919,15.350,152.102
C01213=1097.341,10.097,-54.331,175.921,15.351,152.102
C01214=1097.347,10.347,-54.345,175.923,15.352,152.102
C01215=1097.352,10.597,-54.359,175.925,15.353,152.101
C01216=1097.358,10.846,-54.374,175.927,15.354,152.101
C01217=1097.364,11.096,-54.388,175.929,15.354,152.101
C01218=1097.370,11.346,-54.402,175.931,15.355,152.101
C01219=1097.376,11.594,-54.416,175.934,15.356,152.100
C01220=1097.382,11.844,-54.430,175.936,15.357,152.100
C01221=1097.388,12.094,-54.445,175.938,15.358,152.100
C01222=1097.393,12.343,-54.459,175.939,15.359,152.100
C01223=1097.399,12.593,-54.472,175.941,15.359,152.099
C01224=1097.405,12.843,-54.487,175.944,15.361,152.099
C01225=1097.411,13.092,-54.501,175.946,15.361,152.099
C01226=1097.417,13.341,-54.516,175.948,15.362,152.099
C01227=1097.423,13.591,-54.530,175.950,15.363,152.098
C01228=1097.428,13.841,-54.544,175.952,15.364,152.098
C01229=1097.434,14.090,-54.558,175.954,15.365,152.098
C01230=1097.440,14.340,-54.573,175.956,15.366,152.098
C01231=1097.446,14.589,-54.587,175.958,15.366,152.097
C01232=1097.451,14.839,-54.601,175.961,15.368,152.097
C01233=1097.458,15.088,-54.616,175.962,15.368,152.097
C01234=1097.463,15.361,-54.632,175.964,15.369,152.096
C01235=1097.470,15.633,-54.647,175.967,15.370,152.096
C01236=1097.476,15.906,-54.662,175.969,15.371,152.096
C01237=1097.483,16.179,-54.678,175.972,15.372,152.095
C01238=1097.488,16.428,-54.693,175.974,15.373,152.095
C01239=1097.494,16.677,-54.707,175.976,15.373,152.095
C01240=1097.500,16.927,-54.722,175.978,15.374,152.095
C01241=1097.506,17.176,-54.736,175.980,15.376,152.094
C01242=1097.511,17.426,-54.751,175.982,15.376,152.094
C01243=1097.517,17.676,-54.766,175.984,15.377,152.094
C01244=1097.523,17.925,-54.780,175.986,15.378,152.094
C01245=1097.528,18.174,-54.794,175.989,15.379,152.093
C01246=1097.534,18.424,-54.808,175.990,15.380,152.093
C01247=1097.540,18.673,-54.823,175.992,15.381,152.093
C01248=1097.546,18.923,-54.837,175.994,15.381,152.093
C01249=1097.552,19.173,-54.852,175.997,15.383,152.092
C01250=1097.557,19.422,-54.867,175.999,15.383,152.092
C01251=1097.563,19.671,-54.881,176.001,15.384,152.092
C01252=1097.569,19.921,-54.896,176.002,15.385,152.092
C01253=1097.575,20.170,-54.910,176.005,15.386,152.091
C01254=1097.581,20.420,-54.925,176.007,15.387,152.091
C01255=1097.586,20.670,-54.940,176.009,15.387,152.091
C01256=1097.591,20.919,-54.954,176.012,15.388,152.090
C01257=1097.598,21.169,-54.969,176.014,15.389,152.090
C01258=1097.603,21.418,-54.983,176.016,15.390,152.090
C01259=1097.609,21.668,-54.998,176.018,15.391,152.090
C01260=1097.615,21.917,-55.013,176.020,15.392,152.089
C01261=1097.620,22.166,-55.027,176.022,15.393,152.089
C01262=1097.627,22.416,-55.042,176.024,15.393,152.089
C01263=1097.632,22.666,-55.057,176.026,15.394,152.088
C01264=1097.638,22.915,-55.072,176.029,15.395,152.088
C01265=1097.644,23.164,-55.086,176.030,15.396,152.088
C01266=1097.649,23.414,-55.100,176.032,15.397,152.088
C01267=1097.655,23.664,-55.116,176.034,15.398,152.087
C01268=1097.661,23.913,-55.130,176.037,15.398,152.087
C01269=1097.667,24.163,-55.145,176.039,15.399,152.087
C01270=1097.672,24.412,-55.160,176.041,15.400,152.086
C01271=1097.678,24.662,-55.174,176.044,15.401,152.086
C01272=1097.684,24.911,-55.189,176.045,15.402,152.086
C01273=1097.690,25.160,-55.204,176.047,15.403,152.086
C01274=1097.695,25.410,-55.219,176.049,15.403,152.085
C01275=1097.701,25.660,-55.233,176.052,15.404,152.085
C01276=1097.707,25.909,-55.248,176.054,15.405,152.085
C01277=1097.712,26.158,-55.263,176.056,15.406,152.084
C01278=1097.719,26.408,-55.278,176.059,15.407,152.084
C01279=1097.724,26.657,-55.293,176.060,15.408,152.084
C01280=1097.730,26.907,-55.308,176.062,15.409,152.084
C01281=1097.735,27.157,-55.322,176.065,15.409,152.083
C01282=1097.742,27.406,-55.337,176.067,15.410,152.083
C01283=1097.747,27.656,-55.352,176.069,15.411,152.083
C01284=1097.753,27.905,-55.367,176.071,15.412,152.082
C01285=1097.758,28.154,-55.382,176.074,15.413,152.082
C01286=1097.765,28.404,-55.397,176.076,15.414,152.082
C01287=1097.771,28.653,-55.412,176.078,15.414,152.082
C01288=1097.776,28.903,-55.427,176.080,15.415,152.081
C01289=1097.782,29.152,-55.442,176.082,15.416,152.081
C01290=1097.787,29.403,-55.457,176.084,15.417,152.081
C01291=1097.793,29.652,-55.471,176.086,15.417,152.080
C01292=1097.799,29.901,-55.487,176.089,15.419,152.080
C01293=1097.804,30.150,-55.502,176.091,15.419,152.080
C01294=1097.810,30.400,-55.517,176.093,15.420,152.080
C01295=1097.816,30.649,-55.532,176.095,15.421,152.079
C01296=1097.822,30.899,-55.547,176.097,15.422,152.079
C01297=1097.827,31.148,-55.562,176.099,15.422,152.079
C01298=1097.834,31.422,-55.579,176.102,15.423,152.078
C01299=1097.840,31.696,-55.596,176.104,15.424,152.078
C01300=1097.846,31.970,-55.611,176.107,15.425,152.078
C01301=1097.852,32.244,-55.628,176.109,15.426,152.077
C01302=1097.859,32.493,-55.643,176.112,15.427,152.077
C01303=1097.864,32.743,-55.658,176.113,15.428,152.077
C01304=1097.869,32.993,-55.674,176.116,15.428,152.076
C01305=1097.875,33.241,-55.689,176.118,15.429,152.076
C01306=1097.881,33.491,-55.704,176.120,15.430,152.076
C01307=1097.887,33.740,-55.719,176.122,15.431,152.076
C01308=1097.892,33.990,-55.734,176.124,15.431,152.075
C01309=1097.899,34.240,-55.749,176.127,15.432,152.075
C01310=1097.904,34.489,-55.764,176.129,15.433,152.075
C01311=1097.910,34.739,-55.779,176.131,15.434,152.074
C01312=1097.915,34.988,-55.794,176.134,15.435,152.074
C01313=1097.922,35.237,-55.810,176.136,15.435,152.074
C01314=1097.927,35.487,-55.825,176.137,15.436,152.073
C01315=1097.932,35.737,-55.841,176.140,15.437,152.073
C01316=1097.939,35.986,-55.856,176.142,15.438,152.073
C01317=1097.944,36.235,-55.871,176.144,15.438,152.072
C01318=1097.950,36.485,-55.886,176.147,15.439,152.072
C01319=1097.956,36.735,-55.901,176.149,15.440,152.072
C01320=1097.961,36.984,-55.917,176.151,15.441,152.072
C01321=1097.968,37.233,-55.932,176.154,15.442,152.071
C01322=1097.973,37.483,-55.947,176.156,15.442,152.071
C01323=1097.979,37.732,-55.962,176.158,15.443,152.071
C01324=1097.985,37.982,-55.978,176.161,15.444,152.070
C01325=1097.990,38.231,-55.994,176.162,15.445,152.070
C01326=1097.996,38.481,-56.009,176.164,15.445,152.070
C01327=1098.002,38.730,-56.024,176.167,15.446,152.069
C01328=1098.007,38.980,-56.040,176.169,15.447,152.069
C01329=1098.013,39.229,-56.056,176.171,15.448,152.069
C01330=1098.019,39.478,-56.070,176.174,15.449,152.068
C01331=1098.025,39.728,-56.086,176.176,15.449,152.068
C01332=1098.030,39.977,-56.101,176.178,15.450,152.068
C01333=1098.036,40.227,-56.117,176.181,15.451,152.067
C01334=1098.042,40.476,-56.132,176.183,15.452,152.067
C01335=1098.047,40.726,-56.147,176.185,15.452,152.067
C01336=1098.053,40.976,-56.163,176.188,15.453,152.066
C01337=1098.059,41.225,-56.179,176.189,15.454,152.066
C01338=1098.064,41.474,-56.194,176.191,15.455,152.066
C01339=1098.070,41.724,-56.209,176.194,15.456,152.065
C01340=1098.076,41.973,-56.226,176.196,15.456,152.065
C01341=1098.081,42.222,-56.241,176.198,15.457,152.065
C01342=1098.087,42.472,-56.256,176.201,15.458,152.064
C01343=1098.093,42.721,-56.272,176.203,15.459,152.064
C01344=1098.098,42.971,-56.287,176.205,15.459,152.064
C01345=1098.104,43.220,-56.303,176.208,15.460,152.064
C01346=1098.110,43.470,-56.319,176.210,15.461,152.063
C01347=1098.116,43.719,-56.334,176.212,15.461,152.063
C01348=1098.122,43.968,-56.350,176.214,15.463,152.063
C01349=1098.127,44.218,-56.365,176.217,15.463,152.062
C01350=1098.133,44.467,-56.381,176.219,15.464,152.062
C01351=1098.138,44.717,-56.397,176.222,15.464,152.061
C01352=1098.144,44.967,-56.412,176.223,15.465,152.061
C01353=1098.149,45.216,-56.428,176.225,15.466,152.061
C01354=1098.155,45.466,-56.444,176.228,15.467,152.061
C01355=1098.161,45.715,-56.460,176.230,15.468,152.060
C01356=1098.166,45.964,-56.475,176.233,15.468,152.060
C01357=1098.172,46.213,-56.491,176.235,15.469,152.060
C01358=1098.178,46.463,-56.507,176.237,15.470,152.059
C01359=1098.183,46.712,-56.523,176.240,15.471,152.059
C01360=1098.189,46.962,-56.538,176.242,15.471,152.059
C01361=1098.194,47.211,-56.555,176.244,15.472,152.058
C01362=1098.201,47.486,-56.572,176.247,15.473,152.058
C01363=1098.207,47.760,-56.588,176.250,15.474,152.057
C01364=1098.213,48.033,-56.607,176.252,15.474,152.057
C01365=1098.219,48.307,-56.624,176.254,15.476,152.057
C01366=1098.225,48.557,-56.640,176.257,15.476,152.056
C01367=1098.230,48.806,-56.655,176.259,15.477,152.056
C01368=1098.236,49.055,-56.671,176.261,15.477,152.056
C01369=1098.242,49.305,-56.687,176.263,15.478,152.055
C01370=1098.247,49.555,-56.703,176.266,15.479,152.055
C01371=1098.253,49.803,-56.719,176.268,15.480,152.055
C01372=1098.258,50.053,-56.734,176.270,15.480,152.054
C01373=1098.264,50.303,-56.751,176.273,15.481,152.054
C01374=1098.270,50.552,-56.767,176.275,15.482,152.054
C01375=1098.275,50.801,-56.782,176.277,15.482,152.053
C01376=1098.281,51.051,-56.798,176.280,15.483,152.053
C01377=1098.287,51.300,-56.815,176.282,15.484,152.053
C01378=1098.293,51.550,-56.830,176.285,15.485,152.052
C01379=1098.298,51.799,-56.846,176.287,15.486,152.052
C01380=1098.304,52.048,-56.862,176.289,15.486,152.052
C01381=1098.310,52.298,-56.878,176.292,15.487,152.051
C01382=1098.315,52.548,-56.895,176.294,15.487,152.051
C01383=1098.321,52.797,-56.911,176.296,15.488,152.050
C01384=1098.326,53.046,-56.926,176.299,15.489,152.050
C01385=1098.332,53.296,-56.942,176.301,15.489,152.050
C01386=1098.338,53.545,-56.959,176.304,15.490,152.049
C01387=1098.344,53.794,-56.975,176.306,15.491,152.049
C01388=1098.350,54.044,-56.990,176.308,15.491,152.049
C01389=1098.356,54.294,-57.007,176.311,15.492,152.048
C01390=1098.361,54.542,-57.023,176.313,15.493,152.048
C01391=1098.367,54.792,-57.039,176.316,15.494,152.048
C01392=1098.372,55.042,-57.054,176.318,15.494,152.047
C01393=1098.378,55.291,-57.071,176.320,15.495,152.047
C01394=1098.384,55.541,-57.088,176.323,15.495,152.046
C01395=1098.390,55.790,-57.104,176.325,15.496,152.046
C01396=1098.396,56.039,-57.120,176.327,15.496,152.046
C01397=1098.401,56.289,-57.135,176.330,15.497,152.045
C01398=1098.407,56.538,-57.151,176.332,15.498,152.045
C01399=1098.412,56.787,-57.168,176.335,15.499,152.045
C01400=1098.418,57.037,-57.184,176.337,15.499,152.044
C01401=1098.424,57.286,-57.201,176.339,15.499,152.044
C01402=1098.430,57.536,-57.217,176.342,15.501,152.044
C01403=1098.436,57.785,-57.233,176.344,15.501,152.043
C01404=1098.441,58.035,-57.249,176.347,15.502,152.043
C01405=1098.447,58.284,-57.265,176.349,15.502,152.042
C01406=1098.453,58.534,-57.281,176.351,15.503,152.042
C01407=1098.458,58.783,-57.298,176.354,15.504,152.042
C01408=1098.464,59.032,-57.314,176.356,15.504,152.041
C01409=1098.470,59.281,-57.330,176.358,15.504,152.041
C01410=1098.476,59.531,-57.347,176.361,15.506,152.041
C01411=1098.482,59.780,-57.363,176.363,15.506,152.040
C01412=1098.487,60.029,-57.379,176.366,15.507,152.040
C01413=1098.493,60.279,-57.396,176.368,15.507,152.039
C01414=1098.499,60.528,-57.412,176.370,15.507,152.039
C01415=1098.505,60.778,-57.429,176.373,15.509,152.039
C01416=1098.511,61.027,-57.445,176.375,15.509,152.038
C01417=1098.516,61.277,-57.462,176.378,15.510,152.038
C01418=1098.522,61.526,-57.478,176.380,15.510,152.037
C01419=1098.528,61.775,-57.494,176.383,15.510,152.037
C01420=1098.534,62.025,-57.510,176.386,15.511,152.036
C01421=1098.540,62.274,-57.527,176.388,15.512,152.036
C01422=1098.545,62.524,-57.543,176.390,15.513,152.036
C01423=1098.551,62.773,-57.560,176.393,15.513,152.035
C01424=1098.557,63.022,-57.576,176.395,15.513,152.035
C01425=1098.563,63.272,-57.592,176.398,15.514,152.034
C01426=1098.568,63.546,-57.610,176.400,15.515,152.034
C01427=1098.575,63.820,-57.628,176.403,15.515,152.034
C01428=1098.582,64.093,-57.647,176.406,15.516,152.033
C01429=1098.588,64.366,-57.665,176.408,15.517,152.033
C01430=1098.593,64.616,-57.682,176.411,15.518,152.032
C01431=1098.599,64.865,-57.698,176.413,15.518,152.032
C01432=1098.605,65.115,-57.714,176.416,15.519,152.031
C01433=1098.610,65.364,-57.731,176.418,15.519,152.031
C01434=1098.617,65.613,-57.748,176.421,15.519,152.031
C01435=1098.622,65.863,-57.765,176.424,15.520,152.030
C01436=1098.628,66.112,-57.781,176.426,15.520,152.030
C01437=1098.634,66.361,-57.797,176.428,15.522,152.030
C01438=1098.639,66.611,-57.814,176.431,15.522,152.029
C01439=1098.645,66.860,-57.831,176.434,15.523,152.029
C01440=1098.650,67.110,-57.848,176.436,15.523,152.028
C01441=1098.656,67.359,-57.864,176.438,15.523,152.028
C01442=1098.662,67.609,-57.881,176.441,15.524,152.027
C01443=1098.668,67.858,-57.898,176.443,15.525,152.027
C01444=1098.673,68.108,-57.914,176.446,15.525,152.027
C01445=1098.679,68.356,-57.931,176.448,15.526,152.026
C01446=1098.684,68.606,-57.948,176.450,15.526,152.026
C01447=1098.690,68.855,-57.964,176.453,15.527,152.025
C01448=1098.696,69.105,-57.982,176.456,15.527,152.025
C01449=1098.702,69.354,-57.999,176.459,15.528,152.024
C01450=1098.708,69.604,-58.016,176.461,15.528,152.024
C01451=1098.713,69.853,-58.032,176.464,15.529,152.024
C01452=1098.719,70.102,-58.049,176.466,15.529,152.023
C01453=1098.725,70.352,-58.066,176.468,15.530,152.023
C01454=1098.730,70.601,-58.082,176.471,15.531,152.022
C01455=1098.736,70.850,-58.099,176.473,15.531,152.022
C01456=1098.742,71.100,-58.116,176.476,15.532,152.022
C01457=1098.747,71.349,-58.133,176.478,15.532,152.021
C01458=1098.753,71.598,-58.150,176.481,15.533,152.021
C01459=1098.758,71.848,-58.167,176.483,15.534,152.020
C01460=1098.764,72.097,-58.183,176.486,15.533,152.020
C01461=1098.770,72.346,-58.201,176.489,15.534,152.019
C01462=1098.776,72.597,-58.218,176.491,15.535,152.019
C01463=1098.782,72.845,-58.235,176.494,15.535,152.019
C01464=1098.787,73.095,-58.252,176.496,15.536,152.018
C01465=1098.793,73.344,-58.268,176.499,15.537,152.018
C01466=1098.799,73.593,-58.286,176.501,15.537,152.017
C01467=1098.804,73.843,-58.302,176.504,15.538,152.017
C01468=1098.810,74.092,-58.319,176.506,15.538,152.017
C01469=1098.815,74.341,-58.336,176.509,15.538,152.016
C01470=1098.821,74.590,-58.354,176.511,15.539,152.016
C01471=1098.827,74.841,-58.370,176.514,15.539,152.015
C01472=1098.833,75.090,-58.388,176.517,15.540,152.015
C01473=1098.838,75.339,-58.405,176.519,15.541,152.014
C01474=1098.844,75.588,-58.422,176.522,15.542,152.014
C01475=1098.849,75.838,-58.439,176.524,15.541,152.013
C01476=1098.855,76.087,-58.456,176.526,15.542,152.013
C01477=1098.860,76.336,-58.473,176.529,15.542,152.013
C01478=1098.867,76.586,-58.490,176.532,15.543,152.012
C01479=1098.872,76.835,-58.507,176.535,15.544,152.012
C01480=1098.878,77.084,-58.525,176.537,15.544,152.011
C01481=1098.884,77.334,-58.541,176.540,15.545,152.011
C01482=1098.889,77.583,-58.559,176.542,15.545,152.010
C01483=1098.895,77.833,-58.577,176.545,15.546,152.010
C01484=1098.901,78.082,-58.594,176.547,15.546,152.009
C01485=1098.907,78.331,-58.610,176.550,15.547,152.009
C01486=1098.912,78.581,-58.627,176.553,15.547,152.009
C01487=1098.918,78.830,-58.645,176.555,15.547,152.008
C01488=1098.923,79.079,-58.662,176.558,15.548,152.008
C01489=1098.929,79.329,-58.680,176.560,15.548,152.007
C01490=1098.935,79.602,-58.699,176.563,15.549,152.007
C01491=1098.941,79.875,-58.718,176.566,15.549,152.006
C01492=1098.948,80.149,-58.737,176.569,15.550,152.006
C01493=1098.954,80.423,-58.755,176.572,15.550,152.005
C01494=1098.959,80.672,-58.773,176.575,15.551,152.005
C01495=1098.965,80.922,-58.790,176.577,15.551,152.004
C01496=1098.971,81.171,-58.808,176.579,15.551,152.004
C01497=1098.976,81.421,-58.825,176.582,15.552,152.003
C01498=1098.981,81.670,-58.842,176.584,15.553,152.003
C01499=1098.988,81.918,-58.859,176.588,15.553,152.002
C01500=1098.993,82.169,-58.877,176.590,15.553,152.002
C01501=1098.999,82.418,-58.894,176.593,15.554,152.002
C01502=1099.005,82.667,-58.912,176.595,15.554,152.001
C01503=1099.010,82.916,-58.929,176.598,15.555,152.001
C01504=1099.016,83.166,-58.947,176.600,15.555,152.000
C01505=1099.021,83.415,-58.964,176.603,15.556,152.000
C01506=1099.027,83.664,-58.982,176.606,15.556,151.999
C01507=1099.032,83.913,-58.999,176.609,15.557,151.999
C01508=1099.039,84.163,-59.017,176.611,15.557,151.998
C01509=1099.044,84.413,-59.034,176.614,15.558,151.998
C01510=1099.049,84.662,-59.052,176.617,15.558,151.997
C01511=1099.055,84.911,-59.069,176.619,15.558,151.997
C01512=1099.061,85.160,-59.087,176.622,15.559,151.997
C01513=1099.066,85.410,-59.105,176.624,15.559,151.996
C01514=1099.072,85.659,-59.122,176.627,15.560,151.996
C01515=1099.078,85.908,-59.140,176.630,15.559,151.995
C01516=1099.084,86.158,-59.156,176.633,15.560,151.995
C01517=1099.090,86.407,-59.174,176.635,15.561,151.994
C01518=1099.096,86.656,-59.192,176.638,15.561,151.994
C01519=1099.101,86.905,-59.210,176.640,15.561,151.993
C01520=1099.107,87.155,-59.227,176.643,15.562,151.993
C01521=1099.113,87.404,-59.245,176.646,15.562,151.992
C01522=1099.118,87.653,-59.263,176.649,15.563,151.992
C01523=1099.124,87.902,-59.280,176.651,15.563,151.991
C01524=1099.130,88.152,-59.298,176.654,15.564,151.991
C01525=1099.135,88.401,-59.316,176.657,15.563,151.990
C01526=1099.141,88.650,-59.333,176.660,15.564,151.990
C01527=1099.146,88.900,-59.352,176.662,15.564,151.989
C01528=1099.152,89.149,-59.369,176.664,15.564,151.989
C01529=1099.157,89.398,-59.387,176.667,15.565,151.988
C01530=1099.164,89.648,-59.405,176.670,15.565,151.988
C01531=1099.169,89.897,-59.422,176.673,15.566,151.987
C01532=1099.175,90.147,-59.440,176.675,15.566,151.987
C01533=1099.181,90.396,-59.458,176.678,15.566,151.986
C01534=1099.186,90.645,-59.475,176.681,15.567,151.986
C01535=1099.192,90.895,-59.493,176.684,15.567,151.985
C01536=1099.198,91.144,-59.511,176.686,15.567,151.985
C01537=1099.203,91.393,-59.529,176.689,15.568,151.984
C01538=1099.210,91.642,-59.546,176.691,15.568,151.984
C01539=1099.215,91.891,-59.565,176.695,15.568,151.983
C01540=1099.221,92.141,-59.583,176.697,15.569,151.983
C01541=1099.226,92.390,-59.601,176.700,15.569,151.982
C01542=1099.232,92.639,-59.618,176.702,15.569,151.982
C01543=1099.238,92.889,-59.636,176.706,15.570,151.981
C01544=1099.243,93.138,-59.654,176.708,15.570,151.981
C01545=1099.248,93.387,-59.672,176.711,15.571,151.980
C01546=1099.254,93.637,-59.690,176.713,15.571,151.980
C01547=1099.260,93.885,-59.708,176.717,15.571,151.979
C01548=1099.265,94.135,-59.727,176.719,15.572,151.979
C01549=1099.271,94.384,-59.744,176.722,15.572,151.978
C01550=1099.277,94.633,-59.762,176.724,15.572,151.978
C01551=1099.283,94.883,-59.780,176.727,15.573,151.977
C01552=1099.288,95.132,-59.799,176.730,15.573,151.977
C01553=1099.294,95.382,-59.817,176.733,15.573,151.976
C01554=1099.300,95.656,-59.837,176.735,15.573,151.976
C01555=1099.306,95.928,-59.856,176.739,15.574,151.975
C01556=1099.312,96.203,-59.876,176.742,15.574,151.974
C01557=1099.319,96.476,-59.895,176.745,15.575,151.974
C01558=1099.324,96.725,-59.914,176.747,15.575,151.973
C01559=1099.330,96.975,-59.932,176.751,15.575,151.973
C01560=1099.336,97.224,-59.950,176.753,15.575,151.972
C01561=1099.341,97.473,-59.969,176.756,15.576,151.972
C01562=1099.347,97.722,-59.987,176.759,15.576,151.971
C01563=1099.353,97.972,-60.004,176.762,15.576,151.971
C01564=1099.358,98.221,-60.023,176.764,15.577,151.970
C01565=1099.364,98.471,-60.041,176.767,15.577,151.970
C01566=1099.370,98.720,-60.059,176.770,15.577,151.969
C01567=1099.375,98.969,-60.078,176.773,15.577,151.968
C01568=1099.381,99.218,-60.096,176.775,15.578,151.968
C01569=1099.387,99.468,-60.114,176.779,15.578,151.967
C01570=1099.392,99.717,-60.132,176.781,15.578,151.967
C01571=1099.398,99.966,-60.150,176.784,15.578,151.966
C01572=1099.404,100.215,-60.169,176.787,15.579,151.966
C01573=1099.409,100.465,-60.187,176.790,15.579,151.965
C01574=1099.415,100.713,-60.205,176.792,15.579,151.965
C01575=1099.421,100.963,-60.223,176.796,15.579,151.964
C01576=1099.427,101.213,-60.242,176.798,15.580,151.964
C01577=1099.432,101.461,-60.260,176.801,15.580,151.963
C01578=1099.438,101.712,-60.279,176.804,15.580,151.963
C01579=1099.444,101.960,-60.297,176.807,15.580,151.962
C01580=1099.449,102.210,-60.316,176.809,15.581,151.962
C01581=1099.455,102.458,-60.334,176.812,15.581,151.961
C01582=1099.460,102.708,-60.352,176.815,15.581,151.960
C01583=1099.466,102.957,-60.371,176.818,15.581,151.960
C01584=1099.471,103.207,-60.389,176.820,15.581,151.959
C01585=1099.477,103.455,-60.407,176.823,15.582,151.959
C01586=1099.483,103.705,-60.426,176.826,15.582,151.958
C01587=1099.489,103.954,-60.444,176.829,15.582,151.958
C01588=1099.494,104.203,-60.463,176.832,15.582,151.957
C01589=1099.500,104.452,-60.481,176.835,15.583,151.957
C01590=1099.505,104.702,-60.500,176.837,15.583,151.956
C01591=1099.511,104.952,-60.519,176.840,15.583,151.956
C01592=1099.517,105.200,-60.537,176.843,15.583,151.955
C01593=1099.522,105.450,-60.556,176.846,15.584,151.954
C01594=1099.528,105.699,-60.574,176.849,15.583,151.954
C01595=1099.534,105.948,-60.593,176.852,15.584,151.953
C01596=1099.540,106.198,-60.611,176.854,15.584,151.953
C01597=1099.545,106.447,-60.630,176.858,15.584,151.952
C01598=1099.550,106.696,-60.649,176.861,15.585,151.951
C01599=1099.556,106.945,-60.667,176.863,15.585,151.951
C01600=1099.562,107.194,-60.686,176.866,15.585,151.950
C01601=1099.568,107.444,-60.705,176.869,15.585,151.950
C01602=1099.573,107.693,-60.723,176.872,15.586,151.949
C01603=1099.579,107.942,-60.742,176.875,15.586,151.949
C01604=1099.585,108.191,-60.761,176.878,15.586,151.948
C01605=1099.590,108.440,-60.780,176.880,15.586,151.948
C01606=1099.596,108.690,-60.798,176.884,15.586,151.947
C01607=1099.602,108.939,-60.817,176.886,15.586,151.946
C01608=1099.607,109.188,-60.836,176.889,15.587,151.946
C01609=1099.613,109.437,-60.854,176.892,15.586,151.945
C01610=1099.619,109.687,-60.873,176.895,15.587,151.945
C01611=1099.624,109.936,-60.892,176.898,15.587,151.944
C01612=1099.630,110.185,-60.910,176.901,15.587,151.944
C01613=1099.636,110.435,-60.930,176.903,15.587,151.943
C01614=1099.641,110.683,-60.948,176.907,15.587,151.942
C01615=1099.647,110.933,-60.966,176.909,15.587,151.942
C01616=1099.653,111.183,-60.986,176.913,15.587,151.941
C01617=1099.658,111.431,-61.005,176.916,15.588,151.941
C01618=1099.665,111.705,-61.026,176.919,15.588,151.940
C01619=1099.671,111.979,-61.046,176.922,15.588,151.939
C01620=1099.677,112.253,-61.067,176.925,15.588,151.939
C01621=1099.684,112.526,-61.087,176.929,15.588,151.938
C01622=1099.689,112.776,-61.107,176.931,15.588,151.937
C01623=1099.694,113.024,-61.125,176.934,15.589,151.937
C01624=1099.700,113.274,-61.145,176.937,15.589,151.936
C01625=1099.706,113.523,-61.163,176.940,15.589,151.936
C01626=1099.712,113.772,-61.183,176.943,15.588,151.935
C01627=1099.717,114.021,-61.201,176.946,15.589,151.934
C01628=1099.723,114.270,-61.221,176.949,15.589,151.934
C01629=1099.729,114.520,-61.240,176.952,15.589,151.933
C01630=1099.734,114.768,-61.258,176.954,15.589,151.933
C01631=1099.740,115.018,-61.277,176.958,15.589,151.932
C01632=1099.745,115.268,-61.296,176.961,15.590,151.932
C01633=1099.751,115.517,-61.315,176.963,15.590,151.931
C01634=1099.756,115.766,-61.334,176.967,15.590,151.930
C01635=1099.762,116.015,-61.353,176.970,15.590,151.930
C01636=1099.768,116.264,-61.373,176.973,15.590,151.929
C01637=1099.773,116.513,-61.392,176.975,15.590,151.928
C01638=1099.779,116.762,-61.411,176.979,15.590,151.928
C01639=1099.784,117.012,-61.431,176.981,15.590,151.927
C01640=1099.790,117.261,-61.450,176.984,15.591,151.927
C01641=1099.795,117.510,-61.469,176.988,15.591,151.926
C01642=1099.801,117.759,-61.488,176.990,15.590,151.925
C01643=1099.807,118.009,-61.507,176.994,15.591,151.925
C01644=1099.812,118.258,-61.526,176.996,15.591,151.924
C01645=1099.817,118.507,-61.545,176.999,15.591,151.924
C01646=1099.823,118.756,-61.565,177.002,15.591,151.923
C01647=1099.829,119.006,-61.584,177.005,15.591,151.922
C01648=1099.835,119.255,-61.604,177.008,15.591,151.922
C01649=1099.840,119.504,-61.623,177.011,15.591,151.921
C01650=1099.845,119.753,-61.642,177.014,15.592,151.921
C01651=1099.851,120.002,-61.661,177.017,15.591,151.920
C01652=1099.857,120.252,-61.680,177.021,15.592,151.919
C01653=1099.862,120.501,-61.700,177.023,15.592,151.919
C01654=1099.868,120.750,-61.720,177.027,15.592,151.918
C01655=1099.874,120.999,-61.738,177.029,15.591,151.917
C01656=1099.879,121.248,-61.758,177.032,15.592,151.917
C01657=1099.885,121.498,-61.777,177.035,15.592,151.916
C01658=1099.891,121.746,-61.797,177.038,15.592,151.916
C01659=1099.897,121.996,-61.816,177.042,15.592,151.915
C01660=1099.902,122.245,-61.835,177.044,15.592,151.914
C01661=1099.907,122.494,-61.854,177.048,15.592,151.914
C01662=1099.913,122.743,-61.874,177.050,15.592,151.913
C01663=1099.918,122.993,-61.894,177.054,15.592,151.912
C01664=1099.924,123.242,-61.913,177.056,15.592,151.912
C01665=1099.930,123.491,-61.933,177.060,15.592,151.911
C01666=1099.936,123.740,-61.953,177.062,15.592,151.911
C01667=1099.941,123.990,-61.972,177.066,15.592,151.910
C01668=1099.947,124.238,-61.992,177.069,15.592,151.909
C01669=1099.952,124.487,-62.011,177.072,15.592,151.909
C01670=1099.958,124.737,-62.030,177.075,15.592,151.908
C01671=1099.964,124.985,-62.050,177.078,15.592,151.907
C01672=1099.970,125.235,-62.069,177.081,15.592,151.907
C01673=1099.975,125.484,-62.090,177.084,15.592,151.906
C01674=1099.981,125.733,-62.109,177.087,15.592,151.905
C01675=1099.986,125.983,-62.128,177.091,15.592,151.905
C01676=1099.992,126.232,-62.148,177.093,15.592,151.904
C01677=1099.998,126.481,-62.167,177.097,15.592,151.903
C01678=1100.004,126.730,-62.187,177.099,15.592,151.903
C01679=1100.010,126.979,-62.207,177.103,15.592,151.902
C01680=1100.015,127.228,-62.227,177.105,15.592,151.901
C01681=1100.021,127.478,-62.246,177.109,15.592,151.901
C01682=1100.027,127.751,-62.268,177.112,15.592,151.900
C01683=1100.033,128.025,-62.289,177.116,15.592,151.899
C01684=1100.039,128.299,-62.311,177.119,15.591,151.899
C01685=1100.046,128.572,-62.333,177.122,15.591,151.898
C01686=1100.052,128.822,-62.352,177.126,15.592,151.897
C01687=1100.057,129.071,-62.373,177.128,15.591,151.896
C01688=1100.063,129.320,-62.392,177.132,15.592,151.896
C01689=1100.069,129.569,-62.412,177.134,15.591,151.895
C01690=1100.075,129.818,-62.432,177.138,15.591,151.894
C01691=1100.081,130.067,-62.451,177.141,15.591,151.894
C01692=1100.086,130.316,-62.471,177.144,15.591,151.893
C01693=1100.092,130.566,-62.491,177.148,15.591,151.892
C01694=1100.098,130.815,-62.511,177.150,15.591,151.892
C01695=1100.104,131.064,-62.531,177.154,15.591,151.891
C01696=1100.109,131.313,-62.550,177.156,15.590,151.890
C01697=1100.115,131.562,-62.570,177.160,15.591,151.890
C01698=1100.121,131.811,-62.590,177.163,15.591,151.889
C01699=1100.126,132.060,-62.610,177.166,15.590,151.888
C01700=1100.132,132.309,-62.630,177.169,15.591,151.888
C01701=1100.138,132.558,-62.650,177.172,15.590,151.887
C01702=1100.143,132.808,-62.669,177.176,15.590,151.886
C01703=1100.148,133.057,-62.690,177.179,15.590,151.886
C01704=1100.154,133.306,-62.710,177.182,15.590,151.885
C01705=1100.160,133.555,-62.730,177.185,15.590,151.884
C01706=1100.165,133.804,-62.750,177.188,15.590,151.884
C01707=1100.171,134.053,-62.770,177.191,15.590,151.883
C01708=1100.177,134.302,-62.790,177.194,15.589,151.882
C01709=1100.183,134.551,-62.810,177.197,15.590,151.882
C01710=1100.188,134.801,-62.830,177.201,15.590,151.881
C01711=1100.194,135.050,-62.850,177.204,15.589,151.880
C01712=1100.199,135.299,-62.871,177.207,15.589,151.879
C01713=1100.205,135.548,-62.891,177.210,15.589,151.879
C01714=1100.211,135.797,-62.911,177.213,15.589,151.878
C01715=1100.216,136.047,-62.931,177.217,15.589,151.877
C01716=1100.222,136.296,-62.951,177.220,15.588,151.877
C01717=1100.228,136.545,-62.971,177.223,15.589,151.876
C01718=1100.234,136.793,-62.991,177.226,15.588,151.875
C01719=1100.239,137.043,-63.012,177.229,15.588,151.875
C01720=1100.245,137.291,-63.032,177.233,15.588,151.874
C01721=1100.250,137.541,-63.052,177.236,15.588,151.873
C01722=1100.256,137.791,-63.072,177.239,15.588,151.873
C01723=1100.262,138.040,-63.092,177.242,15.588,151.872
C01724=1100.268,138.289,-63.112,177.245,15.588,151.871
C01725=1100.273,138.538,-63.133,177.248,15.587,151.870
C01726=1100.279,138.787,-63.153,177.252,15.587,151.870
C01727=1100.284,139.036,-63.173,177.255,15.587,151.869
C01728=1100.289,139.285,-63.194,177.258,15.587,151.868
C01729=1100.296,139.534,-63.214,177.261,15.587,151.868
C01730=1100.301,139.783,-63.235,177.264,15.587,151.867
C01731=1100.307,140.032,-63.255,177.268,15.587,151.866
C01732=1100.313,140.281,-63.275,177.271,15.587,151.865
C01733=1100.319,140.530,-63.295,177.274,15.586,151.865
C01734=1100.324,140.779,-63.316,177.278,15.586,151.864
C01735=1100.329,141.028,-63.336,177.280,15.586,151.863
C01736=1100.336,141.278,-63.357,177.284,15.586,151.862
C01737=1100.341,141.527,-63.377,177.287,15.586,151.862
C01738=1100.346,141.776,-63.398,177.290,15.585,151.861
C01739=1100.352,142.025,-63.418,177.294,15.585,151.860
C01740=1100.357,142.274,-63.438,177.296,15.585,151.860
C01741=1100.363,142.523,-63.459,177.300,15.585,151.859
C01742=1100.370,142.772,-63.480,177.304,15.585,151.858
C01743=1100.375,143.021,-63.500,177.306,15.584,151.857
C01744=1100.380,143.270,-63.521,177.310,15.584,151.857
C01745=1100.386,143.519,-63.541,177.313,15.584,151.856
C01746=1100.392,143.793,-63.564,177.316,15.584,151.855
C01747=1100.398,144.067,-63.587,177.320,15.583,151.854
C01748=1100.404,144.340,-63.609,177.324,15.584,151.854
C01749=1100.411,144.613,-63.632,177.327,15.584,151.853
C01750=1100.416,144.863,-63.652,177.331,15.584,151.852
C01751=1100.422,145.112,-63.673,177.334,15.583,151.851
C01752=1100.427,145.361,-63.694,177.338,15.583,151.850
C01753=1100.433,145.610,-63.714,177.340,15.582,151.850
C01754=1100.439,145.859,-63.735,177.344,15.582,151.849
C01755=1100.444,146.108,-63.756,177.348,15.582,151.848
C01756=1100.450,146.358,-63.776,177.350,15.582,151.848
C01757=1100.456,146.607,-63.796,177.354,15.582,151.847
C01758=1100.462,146.855,-63.818,177.357,15.581,151.846
C01759=1100.467,147.105,-63.839,177.360,15.581,151.845
C01760=1100.473,147.354,-63.859,177.364,15.581,151.845
C01761=1100.479,147.602,-63.880,177.367,15.581,151.844
C01762=1100.484,147.851,-63.900,177.370,15.581,151.843
C01763=1100.490,148.101,-63.921,177.373,15.580,151.842
C01764=1100.496,148.350,-63.943,177.377,15.580,151.842
C01765=1100.501,148.599,-63.963,177.380,15.580,151.841
C01766=1100.507,148.849,-63.984,177.383,15.579,151.840
C01767=1100.512,149.097,-64.005,177.387,15.579,151.839
C01768=1100.518,149.346,-64.025,177.390,15.579,151.839
C01769=1100.524,149.596,-64.046,177.393,15.579,151.838
C01770=1100.530,149.844,-64.067,177.397,15.578,151.837
C01771=1100.535,150.093,-64.088,177.400,15.578,151.836
C01772=1100.541,150.342,-64.109,177.403,15.578,151.836
C01773=1100.546,150.592,-64.130,177.407,15.578,151.835
C01774=1100.552,150.840,-64.151,177.410,15.577,151.834
C01775=1100.557,151.089,-64.172,177.413,15.577,151.833
C01776=1100.563,151.339,-64.193,177.417,15.577,151.832
C01777=1100.569,151.588,-64.214,177.420,15.576,151.832
C01778=1100.574,151.837,-64.235,177.424,15.576,151.831
C01779=1100.580,152.086,-64.256,177.426,15.576,151.830
C01780=1100.585,152.335,-64.277,177.430,15.576,151.830
C01781=1100.591,152.584,-64.298,177.434,15.575,151.829
C01782=1100.597,152.833,-64.319,177.437,15.575,151.828
C01783=1100.602,153.082,-64.340,177.440,15.575,151.827
C01784=1100.609,153.331,-64.362,177.444,15.575,151.826
C01785=1100.614,153.580,-64.383,177.447,15.574,151.826
C01786=1100.619,153.829,-64.404,177.450,15.574,151.825
C01787=1100.625,154.079,-64.425,177.453,15.573,151.824
C01788=1100.631,154.327,-64.446,177.457,15.573,151.823
C01789=1100.637,154.577,-64.467,177.461,15.573,151.822
C01790=1100.642,154.825,-64.488,177.463,15.573,151.822
C01791=1100.648,155.074,-64.510,177.467,15.573,151.821
C01792=1100.654,155.324,-64.530,177.471,15.572,151.820
C01793=1100.659,155.572,-64.552,177.474,15.572,151.819
C01794=1100.665,155.821,-64.573,177.477,15.572,151.819
C01795=1100.671,156.071,-64.594,177.480,15.571,151.818
C01796=1100.676,156.319,-64.615,177.484,15.571,151.817
C01797=1100.682,156.568,-64.637,177.487,15.571,151.816
C01798=1100.688,156.817,-64.657,177.490,15.570,151.815
C01799=1100.693,157.067,-64.680,177.494,15.570,151.815
C01800=1100.699,157.315,-64.701,177.498,15.570,151.814
C01801=1100.704,157.565,-64.722,177.501,15.569,151.813
C01802=1100.710,157.814,-64.743,177.504,15.569,151.812
C01803=1100.716,158.062,-64.764,177.508,15.569,151.811
C01804=1100.722,158.311,-64.786,177.511,15.568,151.811
C01805=1100.727,158.561,-64.807,177.515,15.568,151.810
C01806=1100.732,158.810,-64.829,177.518,15.567,151.809
C01807=1100.738,159.059,-64.850,177.521,15.567,151.808
C01808=1100.744,159.308,-64.872,177.525,15.567,151.807
C01809=1100.750,159.556,-64.893,177.528,15.566,151.807
C01810=1100.756,159.830,-64.916,177.532,15.566,151.806
C01811=1100.762,160.104,-64.940,177.536,15.566,151.805
C01812=1100.768,160.377,-64.963,177.539,15.565,151.804
C01813=1100.775,160.650,-64.987,177.543,15.565,151.803
C01814=1100.780,160.898,-65.009,177.547,15.565,151.802
C01815=1100.786,161.148,-65.030,177.550,15.564,151.802
C01816=1100.791,161.397,-65.051,177.554,15.564,151.801
C01817=1100.797,161.646,-65.073,177.557,15.564,151.800
C01818=1100.803,161.895,-65.094,177.560,15.563,151.799
